LIN {X 0,Y 229.274,Z 915.624,A -85,B 0,C 180,E1 -19873.985,E2 -19873.985} C_VEL
LIN {X 0,Y 228.055,Z 917.353,A -85,B 0,C 180,E1 -19875.727,E2 -19875.727} C_VEL
LIN {X 0,Y 226.593,Z 919.668,A -85,B 0,C 180,E1 -19879.275,E2 -19879.275} C_VEL
LIN {X 0,Y 225.973,Z 920.566,A -85,B 0,C 180,E1 -19882.854,E2 -19882.854} C_VEL
LIN {X 0,Y 225.976,Z 920.476,A -85,B 0,C 180,E1 -19884.646,E2 -19884.646} C_VEL
LIN {X 0,Y 225.996,Z 919.977,A -85,B 0,C 180,E1 -19886.434,E2 -19886.434} C_VEL
LIN {X 0,Y 226.528,Z 918.616,A -85,B 0,C 180,E1 -19889.222,E2 -19889.222} C_VEL
LIN {X 0,Y 226.128,Z 920.542,A -85,B 0,C 180,E1 -19891.781,E2 -19891.781} C_VEL
LIN {X 0,Y 225.942,Z 921.419,A -85,B 0,C 180,E1 -19893.567,E2 -19893.567} C_VEL
LIN {X 0,Y 225.888,Z 921.89,A -85,B 0,C 180,E1 -19895.356,E2 -19895.356} C_VEL
LIN {X 0,Y 226.143,Z 921.695,A -85,B 0,C 180,E1 -19898.939,E2 -19898.939} C_VEL
LIN {X 0,Y 227.195,Z 920.074,A -85,B 0,C 180,E1 -19902.506,E2 -19902.506} C_VEL
LIN {X 0,Y 229.242,Z 917.045,A -85,B 0,C 180,E1 -19906.017,E2 -19906.017} C_VEL
LIN {X 0,Y 232.33,Z 912.52,A -85,B 0,C 180,E1 -19909.436,E2 -19909.436} C_VEL
LIN {X 0,Y 235.463,Z 907.702,A -85,B 0,C 180,E1 -19912.195,E2 -19912.195} C_VEL
LIN {X 0,Y 240.567,Z 900.015,A -85,B 0,C 180,E1 -19915.526,E2 -19915.526} C_VEL
LIN {X 0,Y 245.79,Z 891.995,A -85,B 0,C 180,E1 -19918.151,E2 -19918.151} C_VEL
LIN {X 0,Y 250.12,Z 884.192,A -85,B 0,C 180,E1 -19920.383,E2 -19920.383} C_VEL
LIN {X 0,Y 252.409,Z 878.686,A -85,B 0,C 180,E1 -19921.94,E2 -19921.94} C_VEL
LIN {X 0,Y 254.404,Z 871.949,A -85,B 0,C 180,E1 -19924.026,E2 -19924.026} C_VEL
LIN {X 0,Y 255.766,Z 865.461,A -85,B 0,C 180,E1 -19926.236,E2 -19926.236} C_VEL
LIN {X 0,Y 256.678,Z 859.986,A -85,B 0,C 180,E1 -19928.36,E2 -19928.36} C_VEL
LIN {X 0,Y 257.141,Z 856.349,A -85,B 0,C 180,E1 -19930.066,E2 -19930.066} C_VEL
LIN {X 0,Y 257.235,Z 854.79,A -85,B 0,C 180,E1 -19930.974,E2 -19930.974} C_VEL
LIN {X 0,Y 257.299,Z 852.156,A -85,B 0,C 180,E1 -19933.068,E2 -19933.068} C_VEL
LIN {X 0,Y 257.511,Z 850.333,A -85,B 0,C 180,E1 -19935.202,E2 -19935.202} C_VEL
LIN {X 0,Y 257.586,Z 849.784,A -85,B 0,C 180,E1 -19937.449,E2 -19937.449} C_VEL
LIN {X 0,Y 257.795,Z 850.294,A -85,B 0,C 180,E1 -19939.759,E2 -19939.759} C_VEL
LIN {X 0,Y 258.353,Z 851.607,A -85,B 0,C 180,E1 -19942.082,E2 -19942.082} C_VEL
LIN {X 0,Y 258.93,Z 854.139,A -85,B 0,C 180,E1 -19944.516,E2 -19944.516} C_VEL
LIN {X 0,Y 259.161,Z 858.452,A -85,B 0,C 180,E1 -19947.211,E2 -19947.211} C_VEL
LIN {X 0,Y 258.966,Z 861.924,A -85,B 0,C 180,E1 -19948.958,E2 -19948.958} C_VEL
LIN {X 0,Y 258.495,Z 863.102,A -85,B 0,C 180,E1 -19949.349,E2 -19949.349} C_VEL
LIN {X 0,Y 253.364,Z 871.191,A -85,B 0,C 180,E1 -19951.411,E2 -19951.411} C_VEL
LIN {X 0,Y 247.771,Z 879.009,A -85,B 0,C 180,E1 -19953.916,E2 -19953.916} C_VEL
LIN {X 0,Y 243.503,Z 884.513,A -85,B 0,C 180,E1 -19956.166,E2 -19956.166} C_VEL
LIN {X 0,Y 238.668,Z 890.302,A -85,B 0,C 180,E1 -19959.305,E2 -19959.305} C_VEL
LIN {X 0,Y 234.541,Z 894.493,A -85,B 0,C 180,E1 -19962.562,E2 -19962.562} C_VEL
LIN {X 0,Y 231.301,Z 897.237,A -85,B 0,C 180,E1 -19965.93,E2 -19965.93} C_VEL
LIN {X 0,Y 228.992,Z 898.506,A -85,B 0,C 180,E1 -19969.387,E2 -19969.387} C_VEL
LIN {X 0,Y 227.917,Z 898.617,A -85,B 0,C 180,E1 -19971.129,E2 -19971.129} C_VEL
LIN {X 0,Y 226.816,Z 897.718,A -85,B 0,C 180,E1 -19974.665,E2 -19974.665} C_VEL
LIN {X 0,Y 226.441,Z 896.735,A -85,B 0,C 180,E1 -19976.439,E2 -19976.439} C_VEL
LIN {X 0,Y 226.012,Z 893.548,A -85,B 0,C 180,E1 -19979.998,E2 -19979.998} C_VEL
LIN {X 0,Y 225.989,Z 890.103,A -85,B 0,C 180,E1 -19982.672,E2 -19982.672} C_VEL
LIN {X 0,Y 226.162,Z 884.293,A -85,B 0,C 180,E1 -19986.062,E2 -19986.062} C_VEL
LIN {X 0,Y 226.666,Z 877.901,A -85,B 0,C 180,E1 -19988.917,E2 -19988.917} C_VEL
LIN {X 0,Y 227.604,Z 869.128,A -85,B 0,C 180,E1 -19992.028,E2 -19992.028} C_VEL
LIN {X 0,Y 228.751,Z 859.802,A -85,B 0,C 180,E1 -19994.681,E2 -19994.681} C_VEL
LIN {X 0,Y 230.145,Z 849.412,A -85,B 0,C 180,E1 -19997.091,E2 -19997.091} C_VEL
LIN {X 0,Y 231.52,Z 839.174,A -85,B 0,C 180,E1 -19999.044,E2 -19999.044} C_VEL
LIN {X 0,Y 232.891,Z 827.155,A -85,B 0,C 180,E1 -20000.897,E2 -20000.897} C_VEL
LIN {X 0,Y 230.637,Z 814.342,A -85,B 0,C 180,E1 -20002.616,E2 -20002.616} C_VEL
LIN {X 0,Y 228.031,Z 800.57,A -85,B 0,C 180,E1 -20004.085,E2 -20004.085} C_VEL
LIN {X 0,Y 226.663,Z 793.254,A -85,B 0,C 180,E1 -20004.743,E2 -20004.743} C_VEL
LIN {X 0,Y 227.192,Z 793.184,A -85,B 0,C 180,E1 -20009.984,E2 -20009.984} C_VEL
LIN {X 0,Y 227.538,Z 793.139,A -85,B 0,C 180,E1 -20013.775,E2 -20013.775} C_VEL
LIN {X 0,Y 227.764,Z 793.114,A -85,B 0,C 180,E1 -20016.652,E2 -20016.652} C_VEL
LIN {X 0,Y 227.804,Z 793.107,A -85,B 0,C 180,E1 -20020.379,E2 -20020.379} C_VEL
LIN {X 0,Y 227.82,Z 793.106,A -85,B 0,C 180,E1 -20025.193,E2 -20025.193} C_VEL
LIN {X 0,Y 227.819,Z 793.102,A -85,B 0,C 180,E1 -20029.622,E2 -20029.622} C_VEL
LIN {X 0,Y 227.874,Z 793.098,A -85,B 0,C 180,E1 -20034.127,E2 -20034.127} C_VEL
LIN {X 0,Y 227.849,Z 793.098,A -85,B 0,C 180,E1 -20038.374,E2 -20038.374} C_VEL
LIN {X 0,Y 227.848,Z 793.101,A -85,B 0,C 180,E1 -20042.44,E2 -20042.44} C_VEL
LIN {X 0,Y 227.887,Z 793.094,A -85,B 0,C 180,E1 -20046.364,E2 -20046.364} C_VEL
LIN {X 0,Y 227.906,Z 793.094,A -85,B 0,C 180,E1 -20050.171,E2 -20050.171} C_VEL
LIN {X 0,Y 228.012,Z 793.081,A -85,B 0,C 180,E1 -20053.894,E2 -20053.894} C_VEL
LIN {X 0,Y 228.056,Z 793.075,A -85,B 0,C 180,E1 -20057.542,E2 -20057.542} C_VEL
LIN {X 0,Y 228.249,Z 793.052,A -85,B 0,C 180,E1 -20061.144,E2 -20061.144} C_VEL
LIN {X 0,Y 228.296,Z 793.045,A -85,B 0,C 180,E1 -20062.927,E2 -20062.927} C_VEL
LIN {X 0,Y 228.524,Z 793.019,A -85,B 0,C 180,E1 -20068.238,E2 -20068.238} C_VEL
LIN {X 0,Y 228.522,Z 793.019,A -85,B 0,C 180,E1 -20071.762,E2 -20071.762} C_VEL
LIN {X 0,Y 228.295,Z 793.045,A -85,B 0,C 180,E1 -20077.073,E2 -20077.073} C_VEL
LIN {X 0,Y 228.131,Z 793.066,A -85,B 0,C 180,E1 -20080.652,E2 -20080.652} C_VEL
LIN {X 0,Y 228.025,Z 793.079,A -85,B 0,C 180,E1 -20084.275,E2 -20084.275} C_VEL
LIN {X 0,Y 227.943,Z 793.09,A -85,B 0,C 180,E1 -20087.958,E2 -20087.958} C_VEL
LIN {X 0,Y 227.912,Z 793.093,A -85,B 0,C 180,E1 -20092.323,E2 -20092.323} C_VEL
LIN {X 0,Y 227.915,Z 793.096,A -85,B 0,C 180,E1 -20096.593,E2 -20096.593} C_VEL
LIN {X 0,Y 227.866,Z 793.098,A -85,B 0,C 180,E1 -20100.282,E2 -20100.282} C_VEL
LIN {X 0,Y 227.87,Z 793.098,A -85,B 0,C 180,E1 -20103.722,E2 -20103.722} C_VEL
LIN {X 0,Y 227.838,Z 793.101,A -85,B 0,C 180,E1 -20108.093,E2 -20108.093} C_VEL
LIN {X 0,Y 227.8,Z 793.107,A -85,B 0,C 180,E1 -20112.745,E2 -20112.745} C_VEL
LIN {X 0,Y 227.801,Z 793.11,A -85,B 0,C 180,E1 -20117.258,E2 -20117.258} C_VEL
LIN {X 0,Y 227.819,Z 793.105,A -85,B 0,C 180,E1 -20121.907,E2 -20121.907} C_VEL
LIN {X 0,Y 227.769,Z 793.111,A -85,B 0,C 180,E1 -20124.11,E2 -20124.11} C_VEL
LIN {X 0,Y 227.434,Z 793.149,A -85,B 0,C 180,E1 -20128.313,E2 -20128.313} C_VEL
LIN {X 0,Y 226.937,Z 793.215,A -85,B 0,C 180,E1 -20132.322,E2 -20132.322} C_VEL
LIN {X 0,Y 226.654,Z 793.252,A -85,B 0,C 180,E1 -20135.553,E2 -20135.553} C_VEL
LIN {X 0,Y 229.321,Z 806.969,A -85,B 0,C 180,E1 -20136.84,E2 -20136.84} C_VEL
LIN {X 0,Y 231.8,Z 820.663,A -85,B 0,C 180,E1 -20138.474,E2 -20138.474} C_VEL
LIN {X 0,Y 232.666,Z 825.324,A -85,B 0,C 180,E1 -20139.122,E2 -20139.122} C_VEL
LIN {X 0,Y 231.979,Z 833.383,A -85,B 0,C 180,E1 -20140.297,E2 -20140.297} C_VEL
LIN {X 0,Y 230.728,Z 843.502,A -85,B 0,C 180,E1 -20142.039,E2 -20142.039} C_VEL
LIN {X 0,Y 229.496,Z 853.032,A -85,B 0,C 180,E1 -20144.003,E2 -20144.003} C_VEL
LIN {X 0,Y 228.137,Z 863.503,A -85,B 0,C 180,E1 -20146.643,E2 -20146.643} C_VEL
LIN {X 0,Y 227.143,Z 872.111,A -85,B 0,C 180,E1 -20149.303,E2 -20149.303} C_VEL
LIN {X 0,Y 226.404,Z 880.147,A -85,B 0,C 180,E1 -20152.421,E2 -20152.421} C_VEL
LIN {X 0,Y 225.98,Z 886.444,A -85,B 0,C 180,E1 -20155.543,E2 -20155.543} C_VEL
LIN {X 0,Y 225.964,Z 890.617,A -85,B 0,C 180,E1 -20158.22,E2 -20158.22} C_VEL
LIN {X 0,Y 226.118,Z 894.632,A -85,B 0,C 180,E1 -20161.783,E2 -20161.783} C_VEL
LIN {X 0,Y 226.385,Z 896.062,A -85,B 0,C 180,E1 -20163.562,E2 -20163.562} C_VEL
LIN {X 0,Y 227.142,Z 897.716,A -85,B 0,C 180,E1 -20167.111,E2 -20167.111} C_VEL
LIN {X 0,Y 227.829,Z 897.994,A -85,B 0,C 180,E1 -20168.874,E2 -20168.874} C_VEL
LIN {X 0,Y 229.973,Z 897.451,A -85,B 0,C 180,E1 -20172.354,E2 -20172.354} C_VEL
LIN {X 0,Y 231.14,Z 896.64,A -85,B 0,C 180,E1 -20174.08,E2 -20174.08} C_VEL
LIN {X 0,Y 234.297,Z 893.909,A -85,B 0,C 180,E1 -20177.457,E2 -20177.457} C_VEL
LIN {X 0,Y 237.348,Z 890.881,A -85,B 0,C 180,E1 -20179.91,E2 -20179.91} C_VEL
LIN {X 0,Y 242.013,Z 885.458,A -85,B 0,C 180,E1 -20183.083,E2 -20183.083} C_VEL
LIN {X 0,Y 246.059,Z 880.284,A -85,B 0,C 180,E1 -20185.37,E2 -20185.37} C_VEL
LIN {X 0,Y 252.248,Z 871.669,A -85,B 0,C 180,E1 -20188.273,E2 -20188.273} C_VEL
LIN {X 0,Y 257.284,Z 863.741,A -85,B 0,C 180,E1 -20190.356,E2 -20190.356} C_VEL
LIN {X 0,Y 259.094,Z 860.814,A -85,B 0,C 180,E1 -20191.024,E2 -20191.024} C_VEL
LIN {X 0,Y 259.55,Z 858.602,A -85,B 0,C 180,E1 -20191.9,E2 -20191.9} C_VEL
LIN {X 0,Y 259.84,Z 853.152,A -85,B 0,C 180,E1 -20194.612,E2 -20194.612} C_VEL
LIN {X 0,Y 259.696,Z 850.208,A -85,B 0,C 180,E1 -20196.541,E2 -20196.541} C_VEL
LIN {X 0,Y 259.34,Z 848.043,A -85,B 0,C 180,E1 -20198.558,E2 -20198.558} C_VEL
LIN {X 0,Y 258.983,Z 846.706,A -85,B 0,C 180,E1 -20200.64,E2 -20200.64} C_VEL
LIN {X 0,Y 258.907,Z 846.038,A -85,B 0,C 180,E1 -20202.869,E2 -20202.869} C_VEL
LIN {X 0,Y 258.908,Z 846.524,A -85,B 0,C 180,E1 -20205.108,E2 -20205.108} C_VEL
LIN {X 0,Y 258.887,Z 848.218,A -85,B 0,C 180,E1 -20207.26,E2 -20207.26} C_VEL
LIN {X 0,Y 259.001,Z 850.946,A -85,B 0,C 180,E1 -20209.447,E2 -20209.447} C_VEL
LIN {X 0,Y 258.848,Z 853.067,A -85,B 0,C 180,E1 -20210.528,E2 -20210.528} C_VEL
LIN {X 0,Y 257.691,Z 857.975,A -85,B 0,C 180,E1 -20212.273,E2 -20212.273} C_VEL
LIN {X 0,Y 257.305,Z 859.517,A -85,B 0,C 180,E1 -20212.775,E2 -20212.775} C_VEL
LIN {X 0,Y 256.461,Z 861.959,A -85,B 0,C 180,E1 -20213.454,E2 -20213.454} C_VEL
LIN {X 0,Y 253.775,Z 867.478,A -85,B 0,C 180,E1 -20214.607,E2 -20214.607} C_VEL
LIN {X 0,Y 248.764,Z 875.735,A -85,B 0,C 180,E1 -20216.227,E2 -20216.227} C_VEL
LIN {X 0,Y 246.672,Z 879.511,A -85,B 0,C 180,E1 -20217.167,E2 -20217.167} C_VEL
LIN {X 0,Y 246.146,Z 880.683,A -85,B 0,C 180,E1 -20217.516,E2 -20217.516} C_VEL
LIN {X 0,Y 241.237,Z 889.819,A -85,B 0,C 180,E1 -20220.313,E2 -20220.313} C_VEL
LIN {X 0,Y 235.114,Z 898.779,A -85,B 0,C 180,E1 -20223.36,E2 -20223.36} C_VEL
LIN {X 0,Y 229.931,Z 905.805,A -85,B 0,C 180,E1 -20226.491,E2 -20226.491} C_VEL
LIN {X 0,Y 226.613,Z 910.344,A -85,B 0,C 180,E1 -20229.105,E2 -20229.105} C_VEL
LIN {X 0,Y 223.982,Z 913.873,A -85,B 0,C 180,E1 -20231.713,E2 -20231.713} C_VEL
LIN {X 0,Y 221.163,Z 917.308,A -85,B 0,C 180,E1 -20235.273,E2 -20235.273} C_VEL
LIN {X 0,Y 219.602,Z 919.371,A -85,B 0,C 180,E1 -20238.929,E2 -20238.929} C_VEL
LIN {X 0,Y 218.913,Z 919.999,A -85,B 0,C 180,E1 -20242.622,E2 -20242.622} C_VEL
LIN {X 0,Y 218.931,Z 919.755,A -85,B 0,C 180,E1 -20244.474,E2 -20244.474} C_VEL
LIN {X 0,Y 219.283,Z 918.157,A -85,B 0,C 180,E1 -20248.163,E2 -20248.163} C_VEL
LIN {X 0,Y 219.509,Z 917.46,A -85,B 0,C 180,E1 -20249.197,E2 -20249.197} C_VEL
LIN {X 0,Y 219.501,Z 918.235,A -85,B 0,C 180,E1 -20250,E2 -20250} C_VEL
LIN {X 0,Y 218.887,Z 920.572,A -85,B 0,C 180,E1 -20253.682,E2 -20253.682} C_VEL
LIN {X 0,Y 218.826,Z 921.166,A -85,B 0,C 180,E1 -20255.529,E2 -20255.529} C_VEL
LIN {X 0,Y 219.117,Z 921.256,A -85,B 0,C 180,E1 -20259.228,E2 -20259.228} C_VEL
LIN {X 0,Y 220.224,Z 919.881,A -85,B 0,C 180,E1 -20262.908,E2 -20262.908} C_VEL
LIN {X 0,Y 222.421,Z 917.134,A -85,B 0,C 180,E1 -20266.522,E2 -20266.522} C_VEL
LIN {X 0,Y 225.655,Z 913.026,A -85,B 0,C 180,E1 -20270.035,E2 -20270.035} C_VEL
LIN {X 0,Y 228.919,Z 908.548,A -85,B 0,C 180,E1 -20272.828,E2 -20272.828} C_VEL
LIN {X 0,Y 233.583,Z 902.247,A -85,B 0,C 180,E1 -20275.866,E2 -20275.866} C_VEL
LIN {X 0,Y 239.709,Z 893.799,A -85,B 0,C 180,E1 -20278.932,E2 -20278.932} C_VEL
LIN {X 0,Y 244.314,Z 886.391,A -85,B 0,C 180,E1 -20281.184,E2 -20281.184} C_VEL
LIN {X 0,Y 246.853,Z 881.322,A -85,B 0,C 180,E1 -20282.748,E2 -20282.748} C_VEL
LIN {X 0,Y 249.39,Z 874.036,A -85,B 0,C 180,E1 -20285.188,E2 -20285.188} C_VEL
LIN {X 0,Y 251.014,Z 867.959,A -85,B 0,C 180,E1 -20287.482,E2 -20287.482} C_VEL
LIN {X 0,Y 252.24,Z 862.597,A -85,B 0,C 180,E1 -20289.854,E2 -20289.854} C_VEL
LIN {X 0,Y 252.646,Z 860.025,A -85,B 0,C 180,E1 -20291.314,E2 -20291.314} C_VEL
LIN {X 0,Y 252.907,Z 857.226,A -85,B 0,C 180,E1 -20293.736,E2 -20293.736} C_VEL
LIN {X 0,Y 253.184,Z 855.661,A -85,B 0,C 180,E1 -20296.197,E2 -20296.197} C_VEL
LIN {X 0,Y 253.275,Z 855.58,A -85,B 0,C 180,E1 -20298.522,E2 -20298.522} C_VEL
LIN {X 0,Y 253.6,Z 856.404,A -85,B 0,C 180,E1 -20300.893,E2 -20300.893} C_VEL
LIN {X 0,Y 253.997,Z 858.254,A -85,B 0,C 180,E1 -20303.362,E2 -20303.362} C_VEL
LIN {X 0,Y 254.112,Z 860.071,A -85,B 0,C 180,E1 -20304.942,E2 -20304.942} C_VEL
LIN {X 0,Y 253.822,Z 864.506,A -85,B 0,C 180,E1 -20307.704,E2 -20307.704} C_VEL
LIN {X 0,Y 253.671,Z 865.547,A -85,B 0,C 180,E1 -20308.236,E2 -20308.236} C_VEL
LIN {X 0,Y 251.11,Z 869.408,A -85,B 0,C 180,E1 -20309.283,E2 -20309.283} C_VEL
LIN {X 0,Y 244.171,Z 878.647,A -85,B 0,C 180,E1 -20312.112,E2 -20312.112} C_VEL
LIN {X 0,Y 238.725,Z 885.068,A -85,B 0,C 180,E1 -20314.729,E2 -20314.729} C_VEL
LIN {X 0,Y 234.702,Z 889.543,A -85,B 0,C 180,E1 -20317.089,E2 -20317.089} C_VEL
LIN {X 0,Y 229.966,Z 894.111,A -85,B 0,C 180,E1 -20320.354,E2 -20320.354} C_VEL
LIN {X 0,Y 226.128,Z 897.232,A -85,B 0,C 180,E1 -20323.755,E2 -20323.755} C_VEL
LIN {X 0,Y 223.19,Z 898.882,A -85,B 0,C 180,E1 -20327.264,E2 -20327.264} C_VEL
LIN {X 0,Y 220.939,Z 899.166,A -85,B 0,C 180,E1 -20330.847,E2 -20330.847} C_VEL
LIN {X 0,Y 219.752,Z 897.979,A -85,B 0,C 180,E1 -20334.492,E2 -20334.492} C_VEL
LIN {X 0,Y 219.082,Z 895.308,A -85,B 0,C 180,E1 -20338.16,E2 -20338.16} C_VEL
LIN {X 0,Y 218.914,Z 892.292,A -85,B 0,C 180,E1 -20340.918,E2 -20340.918} C_VEL
LIN {X 0,Y 218.944,Z 888.294,A -85,B 0,C 180,E1 -20343.679,E2 -20343.679} C_VEL
LIN {X 0,Y 219.174,Z 882.707,A -85,B 0,C 180,E1 -20346.697,E2 -20346.697} C_VEL
LIN {X 0,Y 219.742,Z 875.83,A -85,B 0,C 180,E1 -20349.664,E2 -20349.664} C_VEL
LIN {X 0,Y 220.652,Z 867.913,A -85,B 0,C 180,E1 -20352.413,E2 -20352.413} C_VEL
LIN {X 0,Y 221.853,Z 858.216,A -85,B 0,C 180,E1 -20355.148,E2 -20355.148} C_VEL
LIN {X 0,Y 223.167,Z 848.457,A -85,B 0,C 180,E1 -20357.406,E2 -20357.406} C_VEL
LIN {X 0,Y 224.565,Z 837.878,A -85,B 0,C 180,E1 -20359.42,E2 -20359.42} C_VEL
LIN {X 0,Y 225.74,Z 828.36,A -85,B 0,C 180,E1 -20360.933,E2 -20360.933} C_VEL
LIN {X 0,Y 225.16,Z 823.7,A -85,B 0,C 180,E1 -20361.618,E2 -20361.618} C_VEL
LIN {X 0,Y 222.678,Z 810.2,A -85,B 0,C 180,E1 -20363.362,E2 -20363.362} C_VEL
LIN {X 0,Y 219.831,Z 795.12,A -85,B 0,C 180,E1 -20364.882,E2 -20364.882} C_VEL
LIN {X 0,Y 219.649,Z 794.127,A -85,B 0,C 180,E1 -20364.987,E2 -20364.987} C_VEL
LIN {X 0,Y 220.183,Z 794.055,A -85,B 0,C 180,E1 -20370.479,E2 -20370.479} C_VEL
LIN {X 0,Y 220.579,Z 794.008,A -85,B 0,C 180,E1 -20374.993,E2 -20374.993} C_VEL
LIN {X 0,Y 220.733,Z 793.987,A -85,B 0,C 180,E1 -20377.251,E2 -20377.251} C_VEL
LIN {X 0,Y 220.768,Z 793.982,A -85,B 0,C 180,E1 -20380.179,E2 -20380.179} C_VEL
LIN {X 0,Y 220.762,Z 793.986,A -85,B 0,C 180,E1 -20384.454,E2 -20384.454} C_VEL
LIN {X 0,Y 220.761,Z 793.982,A -85,B 0,C 180,E1 -20388.045,E2 -20388.045} C_VEL
LIN {X 0,Y 220.8,Z 793.977,A -85,B 0,C 180,E1 -20390.462,E2 -20390.462} C_VEL
LIN {X 0,Y 220.794,Z 793.983,A -85,B 0,C 180,E1 -20395.044,E2 -20395.044} C_VEL
LIN {X 0,Y 220.827,Z 793.976,A -85,B 0,C 180,E1 -20399.388,E2 -20399.388} C_VEL
LIN {X 0,Y 220.868,Z 793.972,A -85,B 0,C 180,E1 -20403.546,E2 -20403.546} C_VEL
LIN {X 0,Y 220.859,Z 793.971,A -85,B 0,C 180,E1 -20407.551,E2 -20407.551} C_VEL
LIN {X 0,Y 220.921,Z 793.964,A -85,B 0,C 180,E1 -20412.617,E2 -20412.617} C_VEL
LIN {X 0,Y 220.993,Z 793.952,A -85,B 0,C 180,E1 -20417.137,E2 -20417.137} C_VEL
LIN {X 0,Y 221.188,Z 793.931,A -85,B 0,C 180,E1 -20420.859,E2 -20420.859} C_VEL
LIN {X 0,Y 221.234,Z 793.924,A -85,B 0,C 180,E1 -20422.7,E2 -20422.7} C_VEL
LIN {X 0,Y 221.458,Z 793.899,A -85,B 0,C 180,E1 -20428.181,E2 -20428.181} C_VEL
LIN {X 0,Y 221.455,Z 793.9,A -85,B 0,C 180,E1 -20431.819,E2 -20431.819} C_VEL
LIN {X 0,Y 221.232,Z 793.924,A -85,B 0,C 180,E1 -20437.3,E2 -20437.3} C_VEL
LIN {X 0,Y 221.052,Z 793.947,A -85,B 0,C 180,E1 -20440.997,E2 -20440.997} C_VEL
LIN {X 0,Y 220.97,Z 793.961,A -85,B 0,C 180,E1 -20446.633,E2 -20446.633} C_VEL
LIN {X 0,Y 220.863,Z 793.974,A -85,B 0,C 180,E1 -20450.489,E2 -20450.489} C_VEL
LIN {X 0,Y 220.84,Z 793.974,A -85,B 0,C 180,E1 -20454.438,E2 -20454.438} C_VEL
LIN {X 0,Y 220.797,Z 793.982,A -85,B 0,C 180,E1 -20458.519,E2 -20458.519} C_VEL
LIN {X 0,Y 220.805,Z 793.978,A -85,B 0,C 180,E1 -20462.758,E2 -20462.758} C_VEL
LIN {X 0,Y 220.804,Z 793.98,A -85,B 0,C 180,E1 -20467.279,E2 -20467.279} C_VEL
LIN {X 0,Y 220.789,Z 793.977,A -85,B 0,C 180,E1 -20470.19,E2 -20470.19} C_VEL
LIN {X 0,Y 220.762,Z 793.984,A -85,B 0,C 180,E1 -20474.457,E2 -20474.457} C_VEL
LIN {X 0,Y 220.761,Z 793.982,A -85,B 0,C 180,E1 -20478.048,E2 -20478.048} C_VEL
LIN {X 0,Y 220.782,Z 793.981,A -85,B 0,C 180,E1 -20482.787,E2 -20482.787} C_VEL
LIN {X 0,Y 220.45,Z 794.023,A -85,B 0,C 180,E1 -20487.185,E2 -20487.185} C_VEL
LIN {X 0,Y 220.261,Z 794.045,A -85,B 0,C 180,E1 -20489.486,E2 -20489.486} C_VEL
LIN {X 0,Y 219.602,Z 794.128,A -85,B 0,C 180,E1 -20495.165,E2 -20495.165} C_VEL
LIN {X 0,Y 219.616,Z 794.127,A -85,B 0,C 180,E1 -20495.324,E2 -20495.324} C_VEL
LIN {X 0,Y 222.387,Z 808.353,A -85,B 0,C 180,E1 -20496.733,E2 -20496.733} C_VEL
LIN {X 0,Y 224.688,Z 821.078,A -85,B 0,C 180,E1 -20498.311,E2 -20498.311} C_VEL
LIN {X 0,Y 225.648,Z 826.797,A -85,B 0,C 180,E1 -20499.128,E2 -20499.128} C_VEL
LIN {X 0,Y 224.175,Z 839.996,A -85,B 0,C 180,E1 -20501.258,E2 -20501.258} C_VEL
LIN {X 0,Y 222.664,Z 851.133,A -85,B 0,C 180,E1 -20503.499,E2 -20503.499} C_VEL
LIN {X 0,Y 221.206,Z 862.094,A -85,B 0,C 180,E1 -20506.217,E2 -20506.217} C_VEL
LIN {X 0,Y 220.165,Z 870.982,A -85,B 0,C 180,E1 -20508.96,E2 -20508.96} C_VEL
LIN {X 0,Y 219.47,Z 878.246,A -85,B 0,C 180,E1 -20511.717,E2 -20511.717} C_VEL
LIN {X 0,Y 218.994,Z 884.18,A -85,B 0,C 180,E1 -20514.477,E2 -20514.477} C_VEL
LIN {X 0,Y 218.884,Z 888.955,A -85,B 0,C 180,E1 -20517.241,E2 -20517.241} C_VEL
LIN {X 0,Y 218.907,Z 892.674,A -85,B 0,C 180,E1 -20520.002,E2 -20520.002} C_VEL
LIN {X 0,Y 219.304,Z 896.122,A -85,B 0,C 180,E1 -20523.677,E2 -20523.677} C_VEL
LIN {X 0,Y 220.121,Z 898.108,A -85,B 0,C 180,E1 -20527.339,E2 -20527.339} C_VEL
LIN {X 0,Y 220.861,Z 898.528,A -85,B 0,C 180,E1 -20529.157,E2 -20529.157} C_VEL
LIN {X 0,Y 223.082,Z 898.252,A -85,B 0,C 180,E1 -20532.742,E2 -20532.742} C_VEL
LIN {X 0,Y 225.932,Z 896.617,A -85,B 0,C 180,E1 -20536.26,E2 -20536.26} C_VEL
LIN {X 0,Y 227.673,Z 895.256,A -85,B 0,C 180,E1 -20537.982,E2 -20537.982} C_VEL
LIN {X 0,Y 232.029,Z 891.365,A -85,B 0,C 180,E1 -20541.315,E2 -20541.315} C_VEL
LIN {X 0,Y 235.758,Z 887.484,A -85,B 0,C 180,E1 -20543.732,E2 -20543.732} C_VEL
LIN {X 0,Y 239.99,Z 882.66,A -85,B 0,C 180,E1 -20546.059,E2 -20546.059} C_VEL
LIN {X 0,Y 245.599,Z 875.726,A -85,B 0,C 180,E1 -20548.642,E2 -20548.642} C_VEL
LIN {X 0,Y 251.649,Z 867.293,A -85,B 0,C 180,E1 -20551.11,E2 -20551.11} C_VEL
LIN {X 0,Y 253.516,Z 864.526,A -85,B 0,C 180,E1 -20551.786,E2 -20551.786} C_VEL
LIN {X 0,Y 254.186,Z 863.241,A -85,B 0,C 180,E1 -20552.173,E2 -20552.173} C_VEL
LIN {X 0,Y 254.792,Z 859.432,A -85,B 0,C 180,E1 -20554.157,E2 -20554.157} C_VEL
LIN {X 0,Y 255.049,Z 855.815,A -85,B 0,C 180,E1 -20556.518,E2 -20556.518} C_VEL
LIN {X 0,Y 254.812,Z 853.129,A -85,B 0,C 180,E1 -20559.441,E2 -20559.441} C_VEL
LIN {X 0,Y 254.667,Z 852.04,A -85,B 0,C 180,E1 -20561.831,E2 -20561.831} C_VEL
LIN {X 0,Y 254.676,Z 851.984,A -85,B 0,C 180,E1 -20564.152,E2 -20564.152} C_VEL
LIN {X 0,Y 254.607,Z 853.265,A -85,B 0,C 180,E1 -20566.363,E2 -20566.363} C_VEL
LIN {X 0,Y 254.625,Z 855.468,A -85,B 0,C 180,E1 -20568.514,E2 -20568.514} C_VEL
LIN {X 0,Y 254.291,Z 857.874,A -85,B 0,C 180,E1 -20569.943,E2 -20569.943} C_VEL
LIN {X 0,Y 252.312,Z 864.065,A -85,B 0,C 180,E1 -20572.208,E2 -20572.208} C_VEL
LIN {X 0,Y 250.105,Z 870.62,A -85,B 0,C 180,E1 -20574.381,E2 -20574.381} C_VEL
LIN {X 0,Y 246.554,Z 879.693,A -85,B 0,C 180,E1 -20577.208,E2 -20577.208} C_VEL
LIN {X 0,Y 246.146,Z 880.683,A -85,B 0,C 180,E1 -20577.516,E2 -20577.516} C_VEL
LIN {X 0,Y 244.869,Z 883.063,A -85,B 0,C 180,E1 -20578.183,E2 -20578.183} C_VEL
LIN {X 0,Y 243.058,Z 885.529,A -85,B 0,C 180,E1 -20578.769,E2 -20578.769} C_VEL
LIN {X 0,Y 238.497,Z 890.44,A -85,B 0,C 180,E1 -20579.802,E2 -20579.802} C_VEL
LIN {X 0,Y 232.457,Z 896.222,A -85,B 0,C 180,E1 -20581.171,E2 -20581.171} C_VEL
LIN {X 0,Y 229.592,Z 899.271,A -85,B 0,C 180,E1 -20582.227,E2 -20582.227} C_VEL
LIN {X 0,Y 224.68,Z 905.316,A -85,B 0,C 180,E1 -20585.022,E2 -20585.022} C_VEL
LIN {X 0,Y 220.004,Z 910.911,A -85,B 0,C 180,E1 -20588.447,E2 -20588.447} C_VEL
LIN {X 0,Y 217.249,Z 914.141,A -85,B 0,C 180,E1 -20591.125,E2 -20591.125} C_VEL
LIN {X 0,Y 214.291,Z 917.274,A -85,B 0,C 180,E1 -20594.789,E2 -20594.789} C_VEL
LIN {X 0,Y 212.609,Z 919,A -85,B 0,C 180,E1 -20598.56,E2 -20598.56} C_VEL
LIN {X 0,Y 211.879,Z 919.346,A -85,B 0,C 180,E1 -20602.376,E2 -20602.376} C_VEL
LIN {X 0,Y 211.897,Z 919.004,A -85,B 0,C 180,E1 -20604.29,E2 -20604.29} C_VEL
LIN {X 0,Y 211.894,Z 918.269,A -85,B 0,C 180,E1 -20606.196,E2 -20606.196} C_VEL
LIN {X 0,Y 212.498,Z 916.413,A -85,B 0,C 180,E1 -20609.289,E2 -20609.289} C_VEL
LIN {X 0,Y 212.063,Z 918.6,A -85,B 0,C 180,E1 -20611.899,E2 -20611.899} C_VEL
LIN {X 0,Y 211.769,Z 920.388,A -85,B 0,C 180,E1 -20615.714,E2 -20615.714} C_VEL
LIN {X 0,Y 212.108,Z 920.715,A -85,B 0,C 180,E1 -20619.536,E2 -20619.536} C_VEL
LIN {X 0,Y 213.268,Z 919.651,A -85,B 0,C 180,E1 -20623.337,E2 -20623.337} C_VEL
LIN {X 0,Y 215.621,Z 917.237,A -85,B 0,C 180,E1 -20627.059,E2 -20627.059} C_VEL
LIN {X 0,Y 218.999,Z 913.416,A -85,B 0,C 180,E1 -20630.671,E2 -20630.671} C_VEL
LIN {X 0,Y 222.105,Z 909.711,A -85,B 0,C 180,E1 -20633.299,E2 -20633.299} C_VEL
LIN {X 0,Y 227.304,Z 903.404,A -85,B 0,C 180,E1 -20636.636,E2 -20636.636} C_VEL
LIN {X 0,Y 232.804,Z 896.597,A -85,B 0,C 180,E1 -20639.378,E2 -20639.378} C_VEL
LIN {X 0,Y 237.777,Z 889.813,A -85,B 0,C 180,E1 -20641.644,E2 -20641.644} C_VEL
LIN {X 0,Y 240.69,Z 884.993,A -85,B 0,C 180,E1 -20643.195,E2 -20643.195} C_VEL
LIN {X 0,Y 243.59,Z 878.502,A -85,B 0,C 180,E1 -20645.512,E2 -20645.512} C_VEL
LIN {X 0,Y 245.561,Z 872.98,A -85,B 0,C 180,E1 -20647.7,E2 -20647.7} C_VEL
LIN {X 0,Y 247.071,Z 868.272,A -85,B 0,C 180,E1 -20649.821,E2 -20649.821} C_VEL
LIN {X 0,Y 247.957,Z 864.793,A -85,B 0,C 180,E1 -20651.905,E2 -20651.905} C_VEL
LIN {X 0,Y 248.132,Z 863.688,A -85,B 0,C 180,E1 -20652.826,E2 -20652.826} C_VEL
LIN {X 0,Y 248.44,Z 861.824,A -85,B 0,C 180,E1 -20655.009,E2 -20655.009} C_VEL
LIN {X 0,Y 248.62,Z 861.016,A -85,B 0,C 180,E1 -20657.305,E2 -20657.305} C_VEL
LIN {X 0,Y 248.747,Z 861.33,A -85,B 0,C 180,E1 -20659.716,E2 -20659.716} C_VEL
LIN {X 0,Y 249,Z 862.533,A -85,B 0,C 180,E1 -20662.214,E2 -20662.214} C_VEL
LIN {X 0,Y 249.099,Z 863.804,A -85,B 0,C 180,E1 -20663.665,E2 -20663.665} C_VEL
LIN {X 0,Y 248.865,Z 866.18,A -85,B 0,C 180,E1 -20665.61,E2 -20665.61} C_VEL
LIN {X 0,Y 248.318,Z 869.042,A -85,B 0,C 180,E1 -20667.468,E2 -20667.468} C_VEL
LIN {X 0,Y 241.815,Z 877.299,A -85,B 0,C 180,E1 -20669.909,E2 -20669.909} C_VEL
LIN {X 0,Y 235.784,Z 884.066,A -85,B 0,C 180,E1 -20672.482,E2 -20672.482} C_VEL
LIN {X 0,Y 231.136,Z 888.806,A -85,B 0,C 180,E1 -20674.804,E2 -20674.804} C_VEL
LIN {X 0,Y 225.847,Z 893.726,A -85,B 0,C 180,E1 -20678.071,E2 -20678.071} C_VEL
LIN {X 0,Y 221.296,Z 897.141,A -85,B 0,C 180,E1 -20681.481,E2 -20681.481} C_VEL
LIN {X 0,Y 217.712,Z 899.197,A -85,B 0,C 180,E1 -20685.032,E2 -20685.032} C_VEL
LIN {X 0,Y 215.105,Z 899.85,A -85,B 0,C 180,E1 -20688.693,E2 -20688.693} C_VEL
LIN {X 0,Y 213.172,Z 899.079,A -85,B 0,C 180,E1 -20692.42,E2 -20692.42} C_VEL
LIN {X 0,Y 212.301,Z 896.889,A -85,B 0,C 180,E1 -20696.202,E2 -20696.202} C_VEL
LIN {X 0,Y 211.911,Z 894.237,A -85,B 0,C 180,E1 -20699.048,E2 -20699.048} C_VEL
LIN {X 0,Y 211.825,Z 890.69,A -85,B 0,C 180,E1 -20701.899,E2 -20701.899} C_VEL
LIN {X 0,Y 211.867,Z 885.787,A -85,B 0,C 180,E1 -20704.954,E2 -20704.954} C_VEL
LIN {X 0,Y 212.358,Z 879.394,A -85,B 0,C 180,E1 -20708.084,E2 -20708.084} C_VEL
LIN {X 0,Y 213.202,Z 870.803,A -85,B 0,C 180,E1 -20711.405,E2 -20711.405} C_VEL
LIN {X 0,Y 214.276,Z 861.752,A -85,B 0,C 180,E1 -20714.238,E2 -20714.238} C_VEL
LIN {X 0,Y 215.83,Z 850.651,A -85,B 0,C 180,E1 -20717.039,E2 -20717.039} C_VEL
LIN {X 0,Y 217.38,Z 839.211,A -85,B 0,C 180,E1 -20719.351,E2 -20719.351} C_VEL
LIN {X 0,Y 218.675,Z 827.665,A -85,B 0,C 180,E1 -20721.246,E2 -20721.246} C_VEL
LIN {X 0,Y 216.347,Z 814.921,A -85,B 0,C 180,E1 -20723.058,E2 -20723.058} C_VEL
LIN {X 0,Y 213.742,Z 800.789,A -85,B 0,C 180,E1 -20724.672,E2 -20724.672} C_VEL
LIN {X 0,Y 212.626,Z 795.001,A -85,B 0,C 180,E1 -20725.251,E2 -20725.251} C_VEL
LIN {X 0,Y 213.175,Z 794.925,A -85,B 0,C 180,E1 -20730.999,E2 -20730.999} C_VEL
LIN {X 0,Y 213.513,Z 794.89,A -85,B 0,C 180,E1 -20734.624,E2 -20734.624} C_VEL
LIN {X 0,Y 213.669,Z 794.868,A -85,B 0,C 180,E1 -20738.676,E2 -20738.676} C_VEL
LIN {X 0,Y 213.698,Z 794.862,A -85,B 0,C 180,E1 -20741.126,E2 -20741.126} C_VEL
LIN {X 0,Y 213.698,Z 794.863,A -85,B 0,C 180,E1 -20743.678,E2 -20743.678} C_VEL
LIN {X 0,Y 213.698,Z 794.865,A -85,B 0,C 180,E1 -20746.343,E2 -20746.343} C_VEL
LIN {X 0,Y 213.711,Z 794.861,A -85,B 0,C 180,E1 -20749.142,E2 -20749.142} C_VEL
LIN {X 0,Y 213.737,Z 794.859,A -85,B 0,C 180,E1 -20753.71,E2 -20753.71} C_VEL
LIN {X 0,Y 213.752,Z 794.853,A -85,B 0,C 180,E1 -20758.26,E2 -20758.26} C_VEL
LIN {X 0,Y 213.781,Z 794.854,A -85,B 0,C 180,E1 -20762.597,E2 -20762.597} C_VEL
LIN {X 0,Y 213.803,Z 794.85,A -85,B 0,C 180,E1 -20766.978,E2 -20766.978} C_VEL
LIN {X 0,Y 213.884,Z 794.841,A -85,B 0,C 180,E1 -20772.799,E2 -20772.799} C_VEL
LIN {X 0,Y 213.932,Z 794.83,A -85,B 0,C 180,E1 -20776.705,E2 -20776.705} C_VEL
LIN {X 0,Y 214.127,Z 794.81,A -85,B 0,C 180,E1 -20780.555,E2 -20780.555} C_VEL
LIN {X 0,Y 214.065,Z 794.816,A -85,B 0,C 180,E1 -20784.348,E2 -20784.348} C_VEL
LIN {X 0,Y 214.395,Z 794.78,A -85,B 0,C 180,E1 -20788.121,E2 -20788.121} C_VEL
LIN {X 0,Y 214.502,Z 794.768,A -85,B 0,C 180,E1 -20790,E2 -20790} C_VEL
LIN {X 0,Y 214.392,Z 794.78,A -85,B 0,C 180,E1 -20791.879,E2 -20791.879} C_VEL
LIN {X 0,Y 214.173,Z 794.804,A -85,B 0,C 180,E1 -20797.542,E2 -20797.542} C_VEL
LIN {X 0,Y 213.983,Z 794.827,A -85,B 0,C 180,E1 -20801.365,E2 -20801.365} C_VEL
LIN {X 0,Y 213.891,Z 794.838,A -85,B 0,C 180,E1 -20805.24,E2 -20805.24} C_VEL
LIN {X 0,Y 213.803,Z 794.851,A -85,B 0,C 180,E1 -20809.191,E2 -20809.191} C_VEL
LIN {X 0,Y 213.795,Z 794.85,A -85,B 0,C 180,E1 -20813.233,E2 -20813.233} C_VEL
LIN {X 0,Y 213.779,Z 794.854,A -85,B 0,C 180,E1 -20817.429,E2 -20817.429} C_VEL
LIN {X 0,Y 213.752,Z 794.853,A -85,B 0,C 180,E1 -20821.74,E2 -20821.74} C_VEL
LIN {X 0,Y 213.737,Z 794.859,A -85,B 0,C 180,E1 -20826.29,E2 -20826.29} C_VEL
LIN {X 0,Y 213.705,Z 794.862,A -85,B 0,C 180,E1 -20831.127,E2 -20831.127} C_VEL
LIN {X 0,Y 213.698,Z 794.865,A -85,B 0,C 180,E1 -20833.681,E2 -20833.681} C_VEL
LIN {X 0,Y 213.698,Z 794.863,A -85,B 0,C 180,E1 -20836.347,E2 -20836.347} C_VEL
LIN {X 0,Y 213.707,Z 794.863,A -85,B 0,C 180,E1 -20839.147,E2 -20839.147} C_VEL
LIN {X 0,Y 213.657,Z 794.871,A -85,B 0,C 180,E1 -20843.697,E2 -20843.697} C_VEL
LIN {X 0,Y 213.516,Z 794.886,A -85,B 0,C 180,E1 -20845.977,E2 -20845.977} C_VEL
LIN {X 0,Y 213.062,Z 794.942,A -85,B 0,C 180,E1 -20850.347,E2 -20850.347} C_VEL
LIN {X 0,Y 212.572,Z 795.004,A -85,B 0,C 180,E1 -20855.076,E2 -20855.076} C_VEL
LIN {X 0,Y 215.162,Z 808.246,A -85,B 0,C 180,E1 -20856.443,E2 -20856.443} C_VEL
LIN {X 0,Y 217.593,Z 821.633,A -85,B 0,C 180,E1 -20858.161,E2 -20858.161} C_VEL
LIN {X 0,Y 218.532,Z 827.825,A -85,B 0,C 180,E1 -20859.083,E2 -20859.083} C_VEL
LIN {X 0,Y 216.907,Z 841.253,A -85,B 0,C 180,E1 -20861.342,E2 -20861.342} C_VEL
LIN {X 0,Y 215.549,Z 851.208,A -85,B 0,C 180,E1 -20863.426,E2 -20863.426} C_VEL
LIN {X 0,Y 214.088,Z 862.138,A -85,B 0,C 180,E1 -20866.234,E2 -20866.234} C_VEL
LIN {X 0,Y 213.043,Z 871.042,A -85,B 0,C 180,E1 -20869.068,E2 -20869.068} C_VEL
LIN {X 0,Y 212.354,Z 878.383,A -85,B 0,C 180,E1 -20871.916,E2 -20871.916} C_VEL
LIN {X 0,Y 211.821,Z 885.176,A -85,B 0,C 180,E1 -20875.193,E2 -20875.193} C_VEL
LIN {X 0,Y 211.787,Z 889.879,A -85,B 0,C 180,E1 -20878.1,E2 -20878.1} C_VEL
LIN {X 0,Y 211.982,Z 894.468,A -85,B 0,C 180,E1 -20881.902,E2 -20881.902} C_VEL
LIN {X 0,Y 212.226,Z 896.176,A -85,B 0,C 180,E1 -20883.799,E2 -20883.799} C_VEL
LIN {X 0,Y 213.087,Z 898.392,A -85,B 0,C 180,E1 -20887.583,E2 -20887.583} C_VEL
LIN {X 0,Y 215.018,Z 899.186,A -85,B 0,C 180,E1 -20891.312,E2 -20891.312} C_VEL
LIN {X 0,Y 217.54,Z 898.557,A -85,B 0,C 180,E1 -20894.98,E2 -20894.98} C_VEL
LIN {X 0,Y 221.054,Z 896.509,A -85,B 0,C 180,E1 -20898.54,E2 -20898.54} C_VEL
LIN {X 0,Y 225.632,Z 893.064,A -85,B 0,C 180,E1 -20901.951,E2 -20901.951} C_VEL
LIN {X 0,Y 230.933,Z 888.108,A -85,B 0,C 180,E1 -20905.22,E2 -20905.22} C_VEL
LIN {X 0,Y 235.539,Z 883.307,A -85,B 0,C 180,E1 -20907.55,E2 -20907.55} C_VEL
LIN {X 0,Y 241.547,Z 876.51,A -85,B 0,C 180,E1 -20910.128,E2 -20910.128} C_VEL
LIN {X 0,Y 248.029,Z 868.186,A -85,B 0,C 180,E1 -20912.575,E2 -20912.575} C_VEL
LIN {X 0,Y 248.943,Z 866.915,A -85,B 0,C 180,E1 -20912.921,E2 -20912.921} C_VEL
LIN {X 0,Y 249.902,Z 862.807,A -85,B 0,C 180,E1 -20915.356,E2 -20915.356} C_VEL
LIN {X 0,Y 250.231,Z 860.689,A -85,B 0,C 180,E1 -20916.94,E2 -20916.94} C_VEL
LIN {X 0,Y 250.18,Z 859.544,A -85,B 0,C 180,E1 -20918.173,E2 -20918.173} C_VEL
LIN {X 0,Y 250.176,Z 858.019,A -85,B 0,C 180,E1 -20920.669,E2 -20920.669} C_VEL
LIN {X 0,Y 250.259,Z 857.489,A -85,B 0,C 180,E1 -20923.1,E2 -20923.1} C_VEL
LIN {X 0,Y 250.214,Z 858.218,A -85,B 0,C 180,E1 -20925.396,E2 -20925.396} C_VEL
LIN {X 0,Y 250.095,Z 860.03,A -85,B 0,C 180,E1 -20927.59,E2 -20927.59} C_VEL
LIN {X 0,Y 249.95,Z 861.303,A -85,B 0,C 180,E1 -20928.597,E2 -20928.597} C_VEL
LIN {X 0,Y 249.406,Z 863.146,A -85,B 0,C 180,E1 -20929.6,E2 -20929.6} C_VEL
LIN {X 0,Y 246.104,Z 871.281,A -85,B 0,C 180,E1 -20932.639,E2 -20932.639} C_VEL
LIN {X 0,Y 242.2,Z 879.959,A -85,B 0,C 180,E1 -20935.577,E2 -20935.577} C_VEL
LIN {X 0,Y 239.011,Z 885.904,A -85,B 0,C 180,E1 -20937.545,E2 -20937.545} C_VEL
LIN {X 0,Y 233.693,Z 893.97,A -85,B 0,C 180,E1 -20940.25,E2 -20940.25} C_VEL
LIN {X 0,Y 229.592,Z 899.271,A -85,B 0,C 180,E1 -20942.227,E2 -20942.227} C_VEL
LIN {X 0,Y 226.808,Z 902.135,A -85,B 0,C 180,E1 -20943.336,E2 -20943.336} C_VEL
LIN {X 0,Y 220.87,Z 906.522,A -85,B 0,C 180,E1 -20945.045,E2 -20945.045} C_VEL
LIN {X 0,Y 215.172,Z 910.217,A -85,B 0,C 180,E1 -20946.919,E2 -20946.919} C_VEL
LIN {X 0,Y 212.816,Z 912.036,A -85,B 0,C 180,E1 -20948.265,E2 -20948.265} C_VEL
LIN {X 0,Y 208.865,Z 915.918,A -85,B 0,C 180,E1 -20952.372,E2 -20952.372} C_VEL
LIN {X 0,Y 206.362,Z 918.027,A -85,B 0,C 180,E1 -20956.208,E2 -20956.208} C_VEL
LIN {X 0,Y 205.095,Z 918.806,A -85,B 0,C 180,E1 -20960.134,E2 -20960.134} C_VEL
LIN {X 0,Y 204.861,Z 918.116,A -85,B 0,C 180,E1 -20964.216,E2 -20964.216} C_VEL
LIN {X 0,Y 205.247,Z 916.071,A -85,B 0,C 180,E1 -20968.038,E2 -20968.038} C_VEL
LIN {X 0,Y 205.525,Z 915.157,A -85,B 0,C 180,E1 -20969.265,E2 -20969.265} C_VEL
LIN {X 0,Y 205.068,Z 917.487,A -85,B 0,C 180,E1 -20971.964,E2 -20971.964} C_VEL
LIN {X 0,Y 204.73,Z 919.557,A -85,B 0,C 180,E1 -20975.911,E2 -20975.911} C_VEL
LIN {X 0,Y 205.088,Z 920.157,A -85,B 0,C 180,E1 -20979.866,E2 -20979.866} C_VEL
LIN {X 0,Y 206.33,Z 919.355,A -85,B 0,C 180,E1 -20983.794,E2 -20983.794} C_VEL
LIN {X 0,Y 208.844,Z 917.24,A -85,B 0,C 180,E1 -20987.63,E2 -20987.63} C_VEL
LIN {X 0,Y 212.376,Z 913.823,A -85,B 0,C 180,E1 -20991.347,E2 -20991.347} C_VEL
LIN {X 0,Y 216.965,Z 909.055,A -85,B 0,C 180,E1 -20994.904,E2 -20994.904} C_VEL
LIN {X 0,Y 222.608,Z 902.851,A -85,B 0,C 180,E1 -20998.266,E2 -20998.266} C_VEL
LIN {X 0,Y 229.457,Z 895.131,A -85,B 0,C 180,E1 -21001.379,E2 -21001.379} C_VEL
LIN {X 0,Y 234.402,Z 888.482,A -85,B 0,C 180,E1 -21003.689,E2 -21003.689} C_VEL
LIN {X 0,Y 236.925,Z 884.069,A -85,B 0,C 180,E1 -21005.341,E2 -21005.341} C_VEL
LIN {X 0,Y 239.627,Z 878.428,A -85,B 0,C 180,E1 -21007.636,E2 -21007.636} C_VEL
LIN {X 0,Y 242.029,Z 872.538,A -85,B 0,C 180,E1 -21010.425,E2 -21010.425} C_VEL
LIN {X 0,Y 243.118,Z 869.229,A -85,B 0,C 180,E1 -21012.645,E2 -21012.645} C_VEL
LIN {X 0,Y 243.346,Z 868.038,A -85,B 0,C 180,E1 -21013.879,E2 -21013.879} C_VEL
LIN {X 0,Y 243.656,Z 866.635,A -85,B 0,C 180,E1 -21016.189,E2 -21016.189} C_VEL
LIN {X 0,Y 243.789,Z 866.344,A -85,B 0,C 180,E1 -21018.55,E2 -21018.55} C_VEL
LIN {X 0,Y 243.913,Z 867.015,A -85,B 0,C 180,E1 -21021.075,E2 -21021.075} C_VEL
LIN {X 0,Y 243.948,Z 868.045,A -85,B 0,C 180,E1 -21022.77,E2 -21022.77} C_VEL
LIN {X 0,Y 243.673,Z 870.014,A -85,B 0,C 180,E1 -21024.77,E2 -21024.77} C_VEL
LIN {X 0,Y 242.928,Z 872.603,A -85,B 0,C 180,E1 -21026.653,E2 -21026.653} C_VEL
LIN {X 0,Y 235.129,Z 881.256,A -85,B 0,C 180,E1 -21029.459,E2 -21029.459} C_VEL
LIN {X 0,Y 229.845,Z 886.539,A -85,B 0,C 180,E1 -21031.708,E2 -21031.708} C_VEL
LIN {X 0,Y 223.54,Z 892.157,A -85,B 0,C 180,E1 -21034.883,E2 -21034.883} C_VEL
LIN {X 0,Y 219.444,Z 895.342,A -85,B 0,C 180,E1 -21037.397,E2 -21037.397} C_VEL
LIN {X 0,Y 214.703,Z 898.44,A -85,B 0,C 180,E1 -21040.891,E2 -21040.891} C_VEL
LIN {X 0,Y 210.935,Z 900.097,A -85,B 0,C 180,E1 -21044.539,E2 -21044.539} C_VEL
LIN {X 0,Y 208.17,Z 900.411,A -85,B 0,C 180,E1 -21048.311,E2 -21048.311} C_VEL
LIN {X 0,Y 206.142,Z 899.367,A -85,B 0,C 180,E1 -21052.16,E2 -21052.16} C_VEL
LIN {X 0,Y 205.225,Z 896.847,A -85,B 0,C 180,E1 -21056.071,E2 -21056.071} C_VEL
LIN {X 0,Y 204.798,Z 892.854,A -85,B 0,C 180,E1 -21059.998,E2 -21059.998} C_VEL
LIN {X 0,Y 204.749,Z 888.736,A -85,B 0,C 180,E1 -21062.949,E2 -21062.949} C_VEL
LIN {X 0,Y 204.9,Z 883.572,A -85,B 0,C 180,E1 -21065.904,E2 -21065.904} C_VEL
LIN {X 0,Y 205.398,Z 877.247,A -85,B 0,C 180,E1 -21068.855,E2 -21068.855} C_VEL
LIN {X 0,Y 206.244,Z 869.476,A -85,B 0,C 180,E1 -21071.796,E2 -21071.796} C_VEL
LIN {X 0,Y 207.388,Z 859.977,A -85,B 0,C 180,E1 -21074.722,E2 -21074.722} C_VEL
LIN {X 0,Y 208.87,Z 849.469,A -85,B 0,C 180,E1 -21077.373,E2 -21077.373} C_VEL
LIN {X 0,Y 210.442,Z 837.758,A -85,B 0,C 180,E1 -21079.761,E2 -21079.761} C_VEL
LIN {X 0,Y 211.505,Z 827.813,A -85,B 0,C 180,E1 -21081.437,E2 -21081.437} C_VEL
LIN {X 0,Y 209.261,Z 815.495,A -85,B 0,C 180,E1 -21083.24,E2 -21083.24} C_VEL
LIN {X 0,Y 206.611,Z 800.915,A -85,B 0,C 180,E1 -21084.952,E2 -21084.952} C_VEL
LIN {X 0,Y 205.579,Z 795.879,A -85,B 0,C 180,E1 -21085.464,E2 -21085.464} C_VEL
LIN {X 0,Y 206.101,Z 795.807,A -85,B 0,C 180,E1 -21090.761,E2 -21090.761} C_VEL
LIN {X 0,Y 206.502,Z 795.76,A -85,B 0,C 180,E1 -21095.347,E2 -21095.347} C_VEL
LIN {X 0,Y 206.635,Z 795.745,A -85,B 0,C 180,E1 -21098.531,E2 -21098.531} C_VEL
LIN {X 0,Y 206.615,Z 795.749,A -85,B 0,C 180,E1 -21102.864,E2 -21102.864} C_VEL
LIN {X 0,Y 206.617,Z 795.746,A -85,B 0,C 180,E1 -21107.133,E2 -21107.133} C_VEL
LIN {X 0,Y 206.682,Z 795.738,A -85,B 0,C 180,E1 -21111.449,E2 -21111.449} C_VEL
LIN {X 0,Y 206.693,Z 795.738,A -85,B 0,C 180,E1 -21114.687,E2 -21114.687} C_VEL
LIN {X 0,Y 206.689,Z 795.737,A -85,B 0,C 180,E1 -21119.333,E2 -21119.333} C_VEL
LIN {X 0,Y 206.698,Z 795.736,A -85,B 0,C 180,E1 -21123.767,E2 -21123.767} C_VEL
LIN {X 0,Y 206.723,Z 795.73,A -85,B 0,C 180,E1 -21128.039,E2 -21128.039} C_VEL
LIN {X 0,Y 206.817,Z 795.721,A -85,B 0,C 180,E1 -21132.191,E2 -21132.191} C_VEL
LIN {X 0,Y 206.871,Z 795.71,A -85,B 0,C 180,E1 -21136.243,E2 -21136.243} C_VEL
LIN {X 0,Y 207.071,Z 795.69,A -85,B 0,C 180,E1 -21140.23,E2 -21140.23} C_VEL
LIN {X 0,Y 207.029,Z 795.693,A -85,B 0,C 180,E1 -21144.155,E2 -21144.155} C_VEL
LIN {X 0,Y 207.334,Z 795.659,A -85,B 0,C 180,E1 -21148.057,E2 -21148.057} C_VEL
LIN {X 0,Y 207.47,Z 795.643,A -85,B 0,C 180,E1 -21150,E2 -21150} C_VEL
LIN {X 0,Y 207.331,Z 795.66,A -85,B 0,C 180,E1 -21151.943,E2 -21151.943} C_VEL
LIN {X 0,Y 207.118,Z 795.684,A -85,B 0,C 180,E1 -21157.801,E2 -21157.801} C_VEL
LIN {X 0,Y 206.906,Z 795.709,A -85,B 0,C 180,E1 -21161.759,E2 -21161.759} C_VEL
LIN {X 0,Y 206.819,Z 795.72,A -85,B 0,C 180,E1 -21165.775,E2 -21165.775} C_VEL
LIN {X 0,Y 206.738,Z 795.731,A -85,B 0,C 180,E1 -21169.874,E2 -21169.874} C_VEL
LIN {X 0,Y 206.731,Z 795.73,A -85,B 0,C 180,E1 -21174.076,E2 -21174.076} C_VEL
LIN {X 0,Y 206.681,Z 795.739,A -85,B 0,C 180,E1 -21178.428,E2 -21178.428} C_VEL
LIN {X 0,Y 206.688,Z 795.737,A -85,B 0,C 180,E1 -21182.96,E2 -21182.96} C_VEL
LIN {X 0,Y 206.673,Z 795.738,A -85,B 0,C 180,E1 -21187.741,E2 -21187.741} C_VEL
LIN {X 0,Y 206.635,Z 795.743,A -85,B 0,C 180,E1 -21191.564,E2 -21191.564} C_VEL
LIN {X 0,Y 206.626,Z 795.746,A -85,B 0,C 180,E1 -21195.584,E2 -21195.584} C_VEL
LIN {X 0,Y 206.648,Z 795.741,A -85,B 0,C 180,E1 -21199.749,E2 -21199.749} C_VEL
LIN {X 0,Y 206.65,Z 795.741,A -85,B 0,C 180,E1 -21202.257,E2 -21202.257} C_VEL
LIN {X 0,Y 206.525,Z 795.757,A -85,B 0,C 180,E1 -21204.757,E2 -21204.757} C_VEL
LIN {X 0,Y 206.168,Z 795.799,A -85,B 0,C 180,E1 -21209.25,E2 -21209.25} C_VEL
LIN {X 0,Y 205.559,Z 795.877,A -85,B 0,C 180,E1 -21214.85,E2 -21214.85} C_VEL
LIN {X 0,Y 208.382,Z 810.451,A -85,B 0,C 180,E1 -21216.451,E2 -21216.451} C_VEL
LIN {X 0,Y 210.75,Z 823.543,A -85,B 0,C 180,E1 -21218.226,E2 -21218.226} C_VEL
LIN {X 0,Y 211.476,Z 827.762,A -85,B 0,C 180,E1 -21218.878,E2 -21218.878} C_VEL
LIN {X 0,Y 209.83,Z 841.049,A -85,B 0,C 180,E1 -21221.195,E2 -21221.195} C_VEL
LIN {X 0,Y 208.452,Z 851.06,A -85,B 0,C 180,E1 -21223.349,E2 -21223.349} C_VEL
LIN {X 0,Y 206.965,Z 862.079,A -85,B 0,C 180,E1 -21226.251,E2 -21226.251} C_VEL
LIN {X 0,Y 205.929,Z 871.104,A -85,B 0,C 180,E1 -21229.183,E2 -21229.183} C_VEL
LIN {X 0,Y 205.209,Z 878.474,A -85,B 0,C 180,E1 -21232.128,E2 -21232.128} C_VEL
LIN {X 0,Y 204.726,Z 884.998,A -85,B 0,C 180,E1 -21235.353,E2 -21235.353} C_VEL
LIN {X 0,Y 204.703,Z 889.367,A -85,B 0,C 180,E1 -21238.035,E2 -21238.035} C_VEL
LIN {X 0,Y 204.812,Z 893.21,A -85,B 0,C 180,E1 -21240.985,E2 -21240.985} C_VEL
LIN {X 0,Y 205.152,Z 896.088,A -85,B 0,C 180,E1 -21243.931,E2 -21243.931} C_VEL
LIN {X 0,Y 206.06,Z 898.658,A -85,B 0,C 180,E1 -21247.843,E2 -21247.843} C_VEL
LIN {X 0,Y 208.094,Z 899.727,A -85,B 0,C 180,E1 -21251.693,E2 -21251.693} C_VEL
LIN {X 0,Y 210.761,Z 899.43,A -85,B 0,C 180,E1 -21255.474,E2 -21255.474} C_VEL
LIN {X 0,Y 214.446,Z 897.783,A -85,B 0,C 180,E1 -21259.133,E2 -21259.133} C_VEL
LIN {X 0,Y 219.234,Z 894.672,A -85,B 0,C 180,E1 -21262.626,E2 -21262.626} C_VEL
LIN {X 0,Y 224.794,Z 890.185,A -85,B 0,C 180,E1 -21265.959,E2 -21265.959} C_VEL
LIN {X 0,Y 229.605,Z 885.8,A -85,B 0,C 180,E1 -21268.325,E2 -21268.325} C_VEL
LIN {X 0,Y 236.76,Z 878.444,A -85,B 0,C 180,E1 -21271.299,E2 -21271.299} C_VEL
LIN {X 0,Y 243.562,Z 870.56,A -85,B 0,C 180,E1 -21273.735,E2 -21273.735} C_VEL
LIN {X 0,Y 244.443,Z 868.286,A -85,B 0,C 180,E1 -21275.103,E2 -21275.103} C_VEL
LIN {X 0,Y 245.156,Z 865.796,A -85,B 0,C 180,E1 -21277.016,E2 -21277.016} C_VEL
LIN {X 0,Y 245.302,Z 864.045,A -85,B 0,C 180,E1 -21279.325,E2 -21279.325} C_VEL
LIN {X 0,Y 245.486,Z 862.985,A -85,B 0,C 180,E1 -21281.896,E2 -21281.896} C_VEL
LIN {X 0,Y 245.596,Z 863.13,A -85,B 0,C 180,E1 -21284.324,E2 -21284.324} C_VEL
LIN {X 0,Y 245.407,Z 864.54,A -85,B 0,C 180,E1 -21286.582,E2 -21286.582} C_VEL
LIN {X 0,Y 245.068,Z 866.274,A -85,B 0,C 180,E1 -21288.215,E2 -21288.215} C_VEL
LIN {X 0,Y 244.191,Z 868.395,A -85,B 0,C 180,E1 -21289.291,E2 -21289.291} C_VEL
LIN {X 0,Y 240.544,Z 875.655,A -85,B 0,C 180,E1 -21292.152,E2 -21292.152} C_VEL
LIN {X 0,Y 236.197,Z 883.638,A -85,B 0,C 180,E1 -21295.056,E2 -21295.056} C_VEL
LIN {X 0,Y 232.575,Z 889.303,A -85,B 0,C 180,E1 -21297.048,E2 -21297.048} C_VEL
LIN {X 0,Y 227.719,Z 895.729,A -85,B 0,C 180,E1 -21299.387,E2 -21299.387} C_VEL
LIN {X 0,Y 221.208,Z 903.163,A -85,B 0,C 180,E1 -21302.569,E2 -21302.569} C_VEL
LIN {X 0,Y 215.795,Z 908.979,A -85,B 0,C 180,E1 -21305.958,E2 -21305.958} C_VEL
LIN {X 0,Y 212.816,Z 912.036,A -85,B 0,C 180,E1 -21308.265,E2 -21308.265} C_VEL
LIN {X 0,Y 210.566,Z 913.685,A -85,B 0,C 180,E1 -21309.679,E2 -21309.679} C_VEL
LIN {X 0,Y 205.475,Z 915.849,A -85,B 0,C 180,E1 -21311.952,E2 -21311.952} C_VEL
LIN {X 0,Y 200.827,Z 917.269,A -85,B 0,C 180,E1 -21314.381,E2 -21314.381} C_VEL
LIN {X 0,Y 199.312,Z 917.75,A -85,B 0,C 180,E1 -21316.004,E2 -21316.004} C_VEL
LIN {X 0,Y 198.091,Z 918.143,A -85,B 0,C 180,E1 -21319.782,E2 -21319.782} C_VEL
LIN {X 0,Y 197.84,Z 917.194,A -85,B 0,C 180,E1 -21324.094,E2 -21324.094} C_VEL
LIN {X 0,Y 198.23,Z 914.904,A -85,B 0,C 180,E1 -21327.968,E2 -21327.968} C_VEL
LIN {X 0,Y 198.543,Z 913.94,A -85,B 0,C 180,E1 -21329.366,E2 -21329.366} C_VEL
LIN {X 0,Y 198.069,Z 916.364,A -85,B 0,C 180,E1 -21332.033,E2 -21332.033} C_VEL
LIN {X 0,Y 197.693,Z 918.627,A -85,B 0,C 180,E1 -21336.122,E2 -21336.122} C_VEL
LIN {X 0,Y 198.084,Z 919.489,A -85,B 0,C 180,E1 -21340.218,E2 -21340.218} C_VEL
LIN {X 0,Y 199.411,Z 919.005,A -85,B 0,C 180,E1 -21344.283,E2 -21344.283} C_VEL
LIN {X 0,Y 202.091,Z 917.238,A -85,B 0,C 180,E1 -21348.239,E2 -21348.239} C_VEL
LIN {X 0,Y 205.786,Z 914.148,A -85,B 0,C 180,E1 -21352.066,E2 -21352.066} C_VEL
LIN {X 0,Y 210.591,Z 909.785,A -85,B 0,C 180,E1 -21355.712,E2 -21355.712} C_VEL
LIN {X 0,Y 216.468,Z 904.08,A -85,B 0,C 180,E1 -21359.144,E2 -21359.144} C_VEL
LIN {X 0,Y 223.583,Z 896.865,A -85,B 0,C 180,E1 -21362.301,E2 -21362.301} C_VEL
LIN {X 0,Y 228.831,Z 890.699,A -85,B 0,C 180,E1 -21364.624,E2 -21364.624} C_VEL
LIN {X 0,Y 231.541,Z 886.6,A -85,B 0,C 180,E1 -21366.291,E2 -21366.291} C_VEL
LIN {X 0,Y 233.82,Z 882.613,A -85,B 0,C 180,E1 -21368.024,E2 -21368.024} C_VEL
LIN {X 0,Y 236.627,Z 877.082,A -85,B 0,C 180,E1 -21370.8,E2 -21370.8} C_VEL
LIN {X 0,Y 237.889,Z 874.159,A -85,B 0,C 180,E1 -21372.804,E2 -21372.804} C_VEL
LIN {X 0,Y 238.383,Z 872.357,A -85,B 0,C 180,E1 -21375.038,E2 -21375.038} C_VEL
LIN {X 0,Y 238.647,Z 871.457,A -85,B 0,C 180,E1 -21377.412,E2 -21377.412} C_VEL
LIN {X 0,Y 238.719,Z 871.588,A -85,B 0,C 180,E1 -21379.948,E2 -21379.948} C_VEL
LIN {X 0,Y 238.685,Z 872.802,A -85,B 0,C 180,E1 -21382.656,E2 -21382.656} C_VEL
LIN {X 0,Y 238.071,Z 874.921,A -85,B 0,C 180,E1 -21384.894,E2 -21384.894} C_VEL
LIN {X 0,Y 237.496,Z 876.061,A -85,B 0,C 180,E1 -21385.787,E2 -21385.787} C_VEL
LIN {X 0,Y 229.439,Z 884.111,A -85,B 0,C 180,E1 -21388.617,E2 -21388.617} C_VEL
LIN {X 0,Y 222.171,Z 890.387,A -85,B 0,C 180,E1 -21391.671,E2 -21391.671} C_VEL
LIN {X 0,Y 215.92,Z 895.121,A -85,B 0,C 180,E1 -21394.965,E2 -21394.965} C_VEL
LIN {X 0,Y 210.489,Z 898.457,A -85,B 0,C 180,E1 -21398.45,E2 -21398.45} C_VEL
LIN {X 0,Y 206.024,Z 900.45,A -85,B 0,C 180,E1 -21402.119,E2 -21402.119} C_VEL
LIN {X 0,Y 202.62,Z 901.115,A -85,B 0,C 180,E1 -21405.946,E2 -21405.946} C_VEL
LIN {X 0,Y 200.006,Z 900.409,A -85,B 0,C 180,E1 -21409.879,E2 -21409.879} C_VEL
LIN {X 0,Y 198.571,Z 898.317,A -85,B 0,C 180,E1 -21413.903,E2 -21413.903} C_VEL
LIN {X 0,Y 197.883,Z 894.797,A -85,B 0,C 180,E1 -21417.963,E2 -21417.963} C_VEL
LIN {X 0,Y 197.704,Z 891.117,A -85,B 0,C 180,E1 -21421.016,E2 -21421.016} C_VEL
LIN {X 0,Y 197.704,Z 885.379,A -85,B 0,C 180,E1 -21424.669,E2 -21424.669} C_VEL
LIN {X 0,Y 198.223,Z 878.008,A -85,B 0,C 180,E1 -21428.316,E2 -21428.316} C_VEL
LIN {X 0,Y 199.134,Z 869.41,A -85,B 0,C 180,E1 -21431.706,E2 -21431.706} C_VEL
LIN {X 0,Y 200.269,Z 859.92,A -85,B 0,C 180,E1 -21434.737,E2 -21434.737} C_VEL
LIN {X 0,Y 201.801,Z 849.284,A -85,B 0,C 180,E1 -21437.478,E2 -21437.478} C_VEL
LIN {X 0,Y 203.397,Z 837.467,A -85,B 0,C 180,E1 -21439.948,E2 -21439.948} C_VEL
LIN {X 0,Y 204.373,Z 828.251,A -85,B 0,C 180,E1 -21441.543,E2 -21441.543} C_VEL
LIN {X 0,Y 202.115,Z 815.872,A -85,B 0,C 180,E1 -21443.422,E2 -21443.422} C_VEL
LIN {X 0,Y 199.577,Z 801.78,A -85,B 0,C 180,E1 -21445.149,E2 -21445.149} C_VEL
LIN {X 0,Y 198.541,Z 796.756,A -85,B 0,C 180,E1 -21445.696,E2 -21445.696} C_VEL
LIN {X 0,Y 198.872,Z 796.71,A -85,B 0,C 180,E1 -21449.651,E2 -21449.651} C_VEL
LIN {X 0,Y 199.159,Z 796.672,A -85,B 0,C 180,E1 -21452.121,E2 -21452.121} C_VEL
LIN {X 0,Y 199.496,Z 796.634,A -85,B 0,C 180,E1 -21456.787,E2 -21456.787} C_VEL
LIN {X 0,Y 199.578,Z 796.62,A -85,B 0,C 180,E1 -21459.332,E2 -21459.332} C_VEL
LIN {X 0,Y 199.564,Z 796.623,A -85,B 0,C 180,E1 -21462.306,E2 -21462.306} C_VEL
LIN {X 0,Y 199.572,Z 796.625,A -85,B 0,C 180,E1 -21465.226,E2 -21465.226} C_VEL
LIN {X 0,Y 199.572,Z 796.622,A -85,B 0,C 180,E1 -21468.003,E2 -21468.003} C_VEL
LIN {X 0,Y 199.604,Z 796.618,A -85,B 0,C 180,E1 -21470.766,E2 -21470.766} C_VEL
LIN {X 0,Y 199.604,Z 796.619,A -85,B 0,C 180,E1 -21475.712,E2 -21475.712} C_VEL
LIN {X 0,Y 199.679,Z 796.606,A -85,B 0,C 180,E1 -21478.133,E2 -21478.133} C_VEL
LIN {X 0,Y 199.636,Z 796.616,A -85,B 0,C 180,E1 -21482.764,E2 -21482.764} C_VEL
LIN {X 0,Y 199.699,Z 796.607,A -85,B 0,C 180,E1 -21487.224,E2 -21487.224} C_VEL
LIN {X 0,Y 199.742,Z 796.604,A -85,B 0,C 180,E1 -21491.798,E2 -21491.798} C_VEL
LIN {X 0,Y 199.808,Z 796.592,A -85,B 0,C 180,E1 -21495.746,E2 -21495.746} C_VEL
LIN {X 0,Y 200.015,Z 796.571,A -85,B 0,C 180,E1 -21499.881,E2 -21499.881} C_VEL
LIN {X 0,Y 199.993,Z 796.57,A -85,B 0,C 180,E1 -21503.948,E2 -21503.948} C_VEL
LIN {X 0,Y 200.276,Z 796.538,A -85,B 0,C 180,E1 -21507.989,E2 -21507.989} C_VEL
LIN {X 0,Y 200.438,Z 796.519,A -85,B 0,C 180,E1 -21510,E2 -21510} C_VEL
LIN {X 0,Y 199.973,Z 796.572,A -85,B 0,C 180,E1 -21514.031,E2 -21514.031} C_VEL
LIN {X 0,Y 200.066,Z 796.564,A -85,B 0,C 180,E1 -21518.078,E2 -21518.078} C_VEL
LIN {X 0,Y 199.856,Z 796.589,A -85,B 0,C 180,E1 -21522.181,E2 -21522.181} C_VEL
LIN {X 0,Y 199.757,Z 796.602,A -85,B 0,C 180,E1 -21526.348,E2 -21526.348} C_VEL
LIN {X 0,Y 199.662,Z 796.613,A -85,B 0,C 180,E1 -21530.61,E2 -21530.61} C_VEL
LIN {X 0,Y 199.643,Z 796.616,A -85,B 0,C 180,E1 -21534.988,E2 -21534.988} C_VEL
LIN {X 0,Y 199.602,Z 796.618,A -85,B 0,C 180,E1 -21539.534,E2 -21539.534} C_VEL
LIN {X 0,Y 199.659,Z 796.609,A -85,B 0,C 180,E1 -21542.354,E2 -21542.354} C_VEL
LIN {X 0,Y 199.617,Z 796.62,A -85,B 0,C 180,E1 -21546.765,E2 -21546.765} C_VEL
LIN {X 0,Y 199.602,Z 796.618,A -85,B 0,C 180,E1 -21549.33,E2 -21549.33} C_VEL
LIN {X 0,Y 199.567,Z 796.622,A -85,B 0,C 180,E1 -21552.311,E2 -21552.311} C_VEL
LIN {X 0,Y 199.572,Z 796.627,A -85,B 0,C 180,E1 -21555.23,E2 -21555.23} C_VEL
LIN {X 0,Y 199.571,Z 796.621,A -85,B 0,C 180,E1 -21558.006,E2 -21558.006} C_VEL
LIN {X 0,Y 199.592,Z 796.618,A -85,B 0,C 180,E1 -21560.774,E2 -21560.774} C_VEL
LIN {X 0,Y 199.49,Z 796.634,A -85,B 0,C 180,E1 -21564.124,E2 -21564.124} C_VEL
LIN {X 0,Y 199.22,Z 796.664,A -85,B 0,C 180,E1 -21568.054,E2 -21568.054} C_VEL
LIN {X 0,Y 198.723,Z 796.729,A -85,B 0,C 180,E1 -21572.631,E2 -21572.631} C_VEL
LIN {X 0,Y 198.538,Z 796.752,A -85,B 0,C 180,E1 -21574.655,E2 -21574.655} C_VEL
LIN {X 0,Y 201.351,Z 811.456,A -85,B 0,C 180,E1 -21576.337,E2 -21576.337} C_VEL
LIN {X 0,Y 203.828,Z 825.117,A -85,B 0,C 180,E1 -21578.291,E2 -21578.291} C_VEL
LIN {X 0,Y 204.34,Z 828.397,A -85,B 0,C 180,E1 -21578.818,E2 -21578.818} C_VEL
LIN {X 0,Y 202.77,Z 840.755,A -85,B 0,C 180,E1 -21581.041,E2 -21581.041} C_VEL
LIN {X 0,Y 201.349,Z 850.895,A -85,B 0,C 180,E1 -21583.266,E2 -21583.266} C_VEL
LIN {X 0,Y 199.847,Z 861.983,A -85,B 0,C 180,E1 -21586.27,E2 -21586.27} C_VEL
LIN {X 0,Y 198.783,Z 871.037,A -85,B 0,C 180,E1 -21589.305,E2 -21589.305} C_VEL
LIN {X 0,Y 197.992,Z 879.574,A -85,B 0,C 180,E1 -21592.865,E2 -21592.865} C_VEL
LIN {X 0,Y 197.652,Z 885.496,A -85,B 0,C 180,E1 -21595.924,E2 -21595.924} C_VEL
LIN {X 0,Y 197.678,Z 890.254,A -85,B 0,C 180,E1 -21598.984,E2 -21598.984} C_VEL
LIN {X 0,Y 197.852,Z 893.974,A -85,B 0,C 180,E1 -21602.038,E2 -21602.038} C_VEL
LIN {X 0,Y 198.081,Z 895.973,A -85,B 0,C 180,E1 -21604.071,E2 -21604.071} C_VEL
LIN {X 0,Y 199.04,Z 898.793,A -85,B 0,C 180,E1 -21608.122,E2 -21608.122} C_VEL
LIN {X 0,Y 201.17,Z 900.222,A -85,B 0,C 180,E1 -21612.102,E2 -21612.102} C_VEL
LIN {X 0,Y 203.998,Z 900.265,A -85,B 0,C 180,E1 -21616,E2 -21616} C_VEL
LIN {X 0,Y 207.853,Z 898.936,A -85,B 0,C 180,E1 -21619.765,E2 -21619.765} C_VEL
LIN {X 0,Y 212.867,Z 896.27,A -85,B 0,C 180,E1 -21623.342,E2 -21623.342} C_VEL
LIN {X 0,Y 218.676,Z 892.215,A -85,B 0,C 180,E1 -21626.742,E2 -21626.742} C_VEL
LIN {X 0,Y 225.458,Z 886.663,A -85,B 0,C 180,E1 -21629.919,E2 -21629.919} C_VEL
LIN {X 0,Y 233.076,Z 879.467,A -85,B 0,C 180,E1 -21632.873,E2 -21632.873} C_VEL
LIN {X 0,Y 238.187,Z 874.123,A -85,B 0,C 180,E1 -21634.612,E2 -21634.612} C_VEL
LIN {X 0,Y 238.757,Z 873.259,A -85,B 0,C 180,E1 -21635.031,E2 -21635.031} C_VEL
LIN {X 0,Y 239.317,Z 872.036,A -85,B 0,C 180,E1 -21635.97,E2 -21635.97} C_VEL
LIN {X 0,Y 240.014,Z 869.996,A -85,B 0,C 180,E1 -21637.947,E2 -21637.947} C_VEL
LIN {X 0,Y 240.363,Z 868.568,A -85,B 0,C 180,E1 -21640.516,E2 -21640.516} C_VEL
LIN {X 0,Y 240.687,Z 868.07,A -85,B 0,C 180,E1 -21643.114,E2 -21643.114} C_VEL
LIN {X 0,Y 240.686,Z 868.393,A -85,B 0,C 180,E1 -21644.493,E2 -21644.493} C_VEL
LIN {X 0,Y 240.59,Z 868.919,A -85,B 0,C 180,E1 -21645.486,E2 -21645.486} C_VEL
LIN {X 0,Y 240.097,Z 870.884,A -85,B 0,C 180,E1 -21647.682,E2 -21647.682} C_VEL
LIN {X 0,Y 238.793,Z 873.306,A -85,B 0,C 180,E1 -21648.911,E2 -21648.911} C_VEL
LIN {X 0,Y 234.935,Z 879.694,A -85,B 0,C 180,E1 -21651.582,E2 -21651.582} C_VEL
LIN {X 0,Y 230.073,Z 887.21,A -85,B 0,C 180,E1 -21654.522,E2 -21654.522} C_VEL
LIN {X 0,Y 225.26,Z 893.493,A -85,B 0,C 180,E1 -21656.907,E2 -21656.907} C_VEL
LIN {X 0,Y 218.274,Z 901.024,A -85,B 0,C 180,E1 -21660.061,E2 -21660.061} C_VEL
LIN {X 0,Y 212.03,Z 907.162,A -85,B 0,C 180,E1 -21663.418,E2 -21663.418} C_VEL
LIN {X 0,Y 206.893,Z 911.878,A -85,B 0,C 180,E1 -21667.005,E2 -21667.005} C_VEL
LIN {X 0,Y 203.826,Z 914.56,A -85,B 0,C 180,E1 -21669.83,E2 -21669.83} C_VEL
LIN {X 0,Y 200.613,Z 916.982,A -85,B 0,C 180,E1 -21673.724,E2 -21673.724} C_VEL
LIN {X 0,Y 199.312,Z 917.75,A -85,B 0,C 180,E1 -21676.004,E2 -21676.004} C_VEL
LIN {X 0,Y 198.023,Z 918.049,A -85,B 0,C 180,E1 -21677.665,E2 -21677.665} C_VEL
LIN {X 0,Y 194.557,Z 917.733,A -85,B 0,C 180,E1 -21680.372,E2 -21680.372} C_VEL
LIN {X 0,Y 191.947,Z 916.856,A -85,B 0,C 180,E1 -21682.59,E2 -21682.59} C_VEL
LIN {X 0,Y 190.895,Z 915.963,A -85,B 0,C 180,E1 -21684.319,E2 -21684.319} C_VEL
LIN {X 0,Y 190.827,Z 915.606,A -85,B 0,C 180,E1 -21684.905,E2 -21684.905} C_VEL
LIN {X 0,Y 191.581,Z 912.551,A -85,B 0,C 180,E1 -21689.343,E2 -21689.343} C_VEL
LIN {X 0,Y 191.083,Z 915.069,A -85,B 0,C 180,E1 -21692.108,E2 -21692.108} C_VEL
LIN {X 0,Y 190.679,Z 917.645,A -85,B 0,C 180,E1 -21696.348,E2 -21696.348} C_VEL
LIN {X 0,Y 191.096,Z 918.784,A -85,B 0,C 180,E1 -21700.596,E2 -21700.596} C_VEL
LIN {X 0,Y 192.514,Z 918.585,A -85,B 0,C 180,E1 -21704.806,E2 -21704.806} C_VEL
LIN {X 0,Y 195.348,Z 917.121,A -85,B 0,C 180,E1 -21708.893,E2 -21708.893} C_VEL
LIN {X 0,Y 199.234,Z 914.418,A -85,B 0,C 180,E1 -21712.832,E2 -21712.832} C_VEL
LIN {X 0,Y 204.264,Z 910.458,A -85,B 0,C 180,E1 -21716.57,E2 -21716.57} C_VEL
LIN {X 0,Y 210.373,Z 905.233,A -85,B 0,C 180,E1 -21720.074,E2 -21720.074} C_VEL
LIN {X 0,Y 217.763,Z 898.561,A -85,B 0,C 180,E1 -21723.275,E2 -21723.275} C_VEL
LIN {X 0,Y 223.276,Z 892.82,A -85,B 0,C 180,E1 -21725.614,E2 -21725.614} C_VEL
LIN {X 0,Y 226.196,Z 889.008,A -85,B 0,C 180,E1 -21727.292,E2 -21727.292} C_VEL
LIN {X 0,Y 228.942,Z 884.863,A -85,B 0,C 180,E1 -21729.317,E2 -21729.317} C_VEL
LIN {X 0,Y 231.704,Z 880.34,A -85,B 0,C 180,E1 -21731.859,E2 -21731.859} C_VEL
LIN {X 0,Y 232.612,Z 878.326,A -85,B 0,C 180,E1 -21733.519,E2 -21733.519} C_VEL
LIN {X 0,Y 233.174,Z 876.614,A -85,B 0,C 180,E1 -21736.334,E2 -21736.334} C_VEL
LIN {X 0,Y 233.332,Z 876.218,A -85,B 0,C 180,E1 -21738.852,E2 -21738.852} C_VEL
LIN {X 0,Y 233.294,Z 876.863,A -85,B 0,C 180,E1 -21741.559,E2 -21741.559} C_VEL
LIN {X 0,Y 233.074,Z 877.607,A -85,B 0,C 180,E1 -21742.908,E2 -21742.908} C_VEL
LIN {X 0,Y 232.118,Z 879.507,A -85,B 0,C 180,E1 -21744.879,E2 -21744.879} C_VEL
LIN {X 0,Y 223.756,Z 886.86,A -85,B 0,C 180,E1 -21747.725,E2 -21747.725} C_VEL
LIN {X 0,Y 218.045,Z 891.3,A -85,B 0,C 180,E1 -21750.025,E2 -21750.025} C_VEL
LIN {X 0,Y 212.805,Z 894.92,A -85,B 0,C 180,E1 -21752.459,E2 -21752.459} C_VEL
LIN {X 0,Y 206.736,Z 898.493,A -85,B 0,C 180,E1 -21755.922,E2 -21755.922} C_VEL
LIN {X 0,Y 201.548,Z 900.784,A -85,B 0,C 180,E1 -21759.59,E2 -21759.59} C_VEL
LIN {X 0,Y 197.407,Z 901.716,A -85,B 0,C 180,E1 -21763.45,E2 -21763.45} C_VEL
LIN {X 0,Y 194.351,Z 901.351,A -85,B 0,C 180,E1 -21767.467,E2 -21767.467} C_VEL
LIN {X 0,Y 192.104,Z 899.657,A -85,B 0,C 180,E1 -21771.583,E2 -21771.583} C_VEL
LIN {X 0,Y 191.084,Z 896.532,A -85,B 0,C 180,E1 -21775.779,E2 -21775.779} C_VEL
LIN {X 0,Y 190.708,Z 893.233,A -85,B 0,C 180,E1 -21778.942,E2 -21778.942} C_VEL
LIN {X 0,Y 190.616,Z 888.984,A -85,B 0,C 180,E1 -21782.111,E2 -21782.111} C_VEL
LIN {X 0,Y 190.756,Z 882.569,A -85,B 0,C 180,E1 -21785.867,E2 -21785.867} C_VEL
LIN {X 0,Y 191.28,Z 875.955,A -85,B 0,C 180,E1 -21788.981,E2 -21788.981} C_VEL
LIN {X 0,Y 192.182,Z 867.792,A -85,B 0,C 180,E1 -21792.136,E2 -21792.136} C_VEL
LIN {X 0,Y 193.414,Z 857.837,A -85,B 0,C 180,E1 -21795.272,E2 -21795.272} C_VEL
LIN {X 0,Y 194.958,Z 846.791,A -85,B 0,C 180,E1 -21798.112,E2 -21798.112} C_VEL
LIN {X 0,Y 196.35,Z 837.172,A -85,B 0,C 180,E1 -21800.149,E2 -21800.149} C_VEL
LIN {X 0,Y 197.324,Z 829.575,A -85,B 0,C 180,E1 -21801.504,E2 -21801.504} C_VEL
LIN {X 0,Y 195.181,Z 817.307,A -85,B 0,C 180,E1 -21803.47,E2 -21803.47} C_VEL
LIN {X 0,Y 192.646,Z 803.149,A -85,B 0,C 180,E1 -21805.294,E2 -21805.294} C_VEL
LIN {X 0,Y 191.53,Z 797.629,A -85,B 0,C 180,E1 -21805.951,E2 -21805.951} C_VEL
LIN {X 0,Y 191.949,Z 797.569,A -85,B 0,C 180,E1 -21810.834,E2 -21810.834} C_VEL
LIN {X 0,Y 192.194,Z 797.541,A -85,B 0,C 180,E1 -21813.262,E2 -21813.262} C_VEL
LIN {X 0,Y 192.461,Z 797.512,A -85,B 0,C 180,E1 -21816.547,E2 -21816.547} C_VEL
LIN {X 0,Y 192.498,Z 797.503,A -85,B 0,C 180,E1 -21821.081,E2 -21821.081} C_VEL
LIN {X 0,Y 192.484,Z 797.507,A -85,B 0,C 180,E1 -21826.074,E2 -21826.074} C_VEL
LIN {X 0,Y 192.511,Z 797.499,A -85,B 0,C 180,E1 -21830.05,E2 -21830.05} C_VEL
LIN {X 0,Y 192.554,Z 797.498,A -85,B 0,C 180,E1 -21834.269,E2 -21834.269} C_VEL
LIN {X 0,Y 192.598,Z 797.492,A -85,B 0,C 180,E1 -21837.059,E2 -21837.059} C_VEL
LIN {X 0,Y 192.613,Z 797.491,A -85,B 0,C 180,E1 -21841.684,E2 -21841.684} C_VEL
LIN {X 0,Y 192.671,Z 797.48,A -85,B 0,C 180,E1 -21846.344,E2 -21846.344} C_VEL
LIN {X 0,Y 192.69,Z 797.484,A -85,B 0,C 180,E1 -21851.487,E2 -21851.487} C_VEL
LIN {X 0,Y 192.733,Z 797.475,A -85,B 0,C 180,E1 -21855.211,E2 -21855.211} C_VEL
LIN {X 0,Y 192.937,Z 797.451,A -85,B 0,C 180,E1 -21859.566,E2 -21859.566} C_VEL
LIN {X 0,Y 192.957,Z 797.448,A -85,B 0,C 180,E1 -21863.727,E2 -21863.727} C_VEL
LIN {X 0,Y 193.221,Z 797.416,A -85,B 0,C 180,E1 -21867.916,E2 -21867.916} C_VEL
LIN {X 0,Y 193.404,Z 797.395,A -85,B 0,C 180,E1 -21870,E2 -21870} C_VEL
LIN {X 0,Y 192.921,Z 797.45,A -85,B 0,C 180,E1 -21874.178,E2 -21874.178} C_VEL
LIN {X 0,Y 193.017,Z 797.443,A -85,B 0,C 180,E1 -21878.375,E2 -21878.375} C_VEL
LIN {X 0,Y 192.782,Z 797.466,A -85,B 0,C 180,E1 -21882.635,E2 -21882.635} C_VEL
LIN {X 0,Y 192.711,Z 797.479,A -85,B 0,C 180,E1 -21886.963,E2 -21886.963} C_VEL
LIN {X 0,Y 192.598,Z 797.489,A -85,B 0,C 180,E1 -21891.402,E2 -21891.402} C_VEL
LIN {X 0,Y 192.632,Z 797.486,A -85,B 0,C 180,E1 -21894.209,E2 -21894.209} C_VEL
LIN {X 0,Y 192.595,Z 797.494,A -85,B 0,C 180,E1 -21898.867,E2 -21898.867} C_VEL
LIN {X 0,Y 192.588,Z 797.495,A -85,B 0,C 180,E1 -21903.188,E2 -21903.188} C_VEL
LIN {X 0,Y 192.545,Z 797.498,A -85,B 0,C 180,E1 -21908.354,E2 -21908.354} C_VEL
LIN {X 0,Y 192.484,Z 797.508,A -85,B 0,C 180,E1 -21913.097,E2 -21913.097} C_VEL
LIN {X 0,Y 192.484,Z 797.508,A -85,B 0,C 180,E1 -21916.907,E2 -21916.907} C_VEL
LIN {X 0,Y 192.492,Z 797.507,A -85,B 0,C 180,E1 -21921.637,E2 -21921.637} C_VEL
LIN {X 0,Y 192.428,Z 797.514,A -85,B 0,C 180,E1 -21924.245,E2 -21924.245} C_VEL
LIN {X 0,Y 192.012,Z 797.561,A -85,B 0,C 180,E1 -21929.177,E2 -21929.177} C_VEL
LIN {X 0,Y 191.52,Z 797.627,A -85,B 0,C 180,E1 -21934.355,E2 -21934.355} C_VEL
LIN {X 0,Y 191.522,Z 797.713,A -85,B 0,C 180,E1 -21934.475,E2 -21934.475} C_VEL
LIN {X 0,Y 194.104,Z 811.265,A -85,B 0,C 180,E1 -21936.06,E2 -21936.06} C_VEL
LIN {X 0,Y 196.415,Z 824.156,A -85,B 0,C 180,E1 -21937.939,E2 -21937.939} C_VEL
LIN {X 0,Y 197.162,Z 828.296,A -85,B 0,C 180,E1 -21938.629,E2 -21938.629} C_VEL
LIN {X 0,Y 195.713,Z 840.407,A -85,B 0,C 180,E1 -21940.875,E2 -21940.875} C_VEL
LIN {X 0,Y 194.143,Z 851.593,A -85,B 0,C 180,E1 -21943.439,E2 -21943.439} C_VEL
LIN {X 0,Y 192.748,Z 861.708,A -85,B 0,C 180,E1 -21946.293,E2 -21946.293} C_VEL
LIN {X 0,Y 191.683,Z 870.91,A -85,B 0,C 180,E1 -21949.439,E2 -21949.439} C_VEL
LIN {X 0,Y 190.985,Z 878.452,A -85,B 0,C 180,E1 -21952.602,E2 -21952.602} C_VEL
LIN {X 0,Y 190.587,Z 884.581,A -85,B 0,C 180,E1 -21955.773,E2 -21955.773} C_VEL
LIN {X 0,Y 190.612,Z 889.594,A -85,B 0,C 180,E1 -21958.946,E2 -21958.946} C_VEL
LIN {X 0,Y 190.789,Z 893.592,A -85,B 0,C 180,E1 -21962.113,E2 -21962.113} C_VEL
LIN {X 0,Y 191.4,Z 897.472,A -85,B 0,C 180,E1 -21966.326,E2 -21966.326} C_VEL
LIN {X 0,Y 192.984,Z 899.939,A -85,B 0,C 180,E1 -21970.493,E2 -21970.493} C_VEL
LIN {X 0,Y 195.625,Z 900.974,A -85,B 0,C 180,E1 -21974.567,E2 -21974.567} C_VEL
LIN {X 0,Y 199.141,Z 900.699,A -85,B 0,C 180,E1 -21978.521,E2 -21978.521} C_VEL
LIN {X 0,Y 201.28,Z 900.082,A -85,B 0,C 180,E1 -21980.438,E2 -21980.438} C_VEL
LIN {X 0,Y 206.534,Z 897.781,A -85,B 0,C 180,E1 -21984.103,E2 -21984.103} C_VEL
LIN {X 0,Y 212.603,Z 894.158,A -85,B 0,C 180,E1 -21987.57,E2 -21987.57} C_VEL
LIN {X 0,Y 217.795,Z 890.526,A -85,B 0,C 180,E1 -21990.013,E2 -21990.013} C_VEL
LIN {X 0,Y 225.543,Z 884.344,A -85,B 0,C 180,E1 -21993.047,E2 -21993.047} C_VEL
LIN {X 0,Y 231.734,Z 878.67,A -85,B 0,C 180,E1 -21995.188,E2 -21995.188} C_VEL
LIN {X 0,Y 233.55,Z 876.781,A -85,B 0,C 180,E1 -21995.932,E2 -21995.932} C_VEL
LIN {X 0,Y 234.102,Z 875.756,A -85,B 0,C 180,E1 -21996.902,E2 -21996.902} C_VEL
LIN {X 0,Y 234.802,Z 874.176,A -85,B 0,C 180,E1 -21998.946,E2 -21998.946} C_VEL
LIN {X 0,Y 235.328,Z 873.112,A -85,B 0,C 180,E1 -22001.701,E2 -22001.701} C_VEL
LIN {X 0,Y 235.559,Z 873.038,A -85,B 0,C 180,E1 -22003.333,E2 -22003.333} C_VEL
LIN {X 0,Y 235.565,Z 873.252,A -85,B 0,C 180,E1 -22004.272,E2 -22004.272} C_VEL
LIN {X 0,Y 235.105,Z 874.769,A -85,B 0,C 180,E1 -22006.564,E2 -22006.564} C_VEL
LIN {X 0,Y 234.261,Z 876.403,A -85,B 0,C 180,E1 -22007.769,E2 -22007.769} C_VEL
LIN {X 0,Y 230.516,Z 881.687,A -85,B 0,C 180,E1 -22010.189,E2 -22010.189} C_VEL
LIN {X 0,Y 226.187,Z 887.561,A -85,B 0,C 180,E1 -22012.706,E2 -22012.706} C_VEL
LIN {X 0,Y 221.302,Z 893.452,A -85,B 0,C 180,E1 -22015.136,E2 -22015.136} C_VEL
LIN {X 0,Y 215.923,Z 899.013,A -85,B 0,C 180,E1 -22017.517,E2 -22017.517} C_VEL
LIN {X 0,Y 208.872,Z 905.33,A -85,B 0,C 180,E1 -22020.798,E2 -22020.798} C_VEL
LIN {X 0,Y 204.063,Z 909.357,A -85,B 0,C 180,E1 -22023.57,E2 -22023.57} C_VEL
LIN {X 0,Y 199.237,Z 913.145,A -85,B 0,C 180,E1 -22027.169,E2 -22027.169} C_VEL
LIN {X 0,Y 195.364,Z 915.845,A -85,B 0,C 180,E1 -22031.109,E2 -22031.109} C_VEL
LIN {X 0,Y 192.542,Z 917.294,A -85,B 0,C 180,E1 -22035.196,E2 -22035.196} C_VEL
LIN {X 0,Y 191.103,Z 917.454,A -85,B 0,C 180,E1 -22039.404,E2 -22039.404} C_VEL
LIN {X 0,Y 190.826,Z 916.128,A -85,B 0,C 180,E1 -22043.946,E2 -22043.946} C_VEL
LIN {X 0,Y 190.827,Z 915.606,A -85,B 0,C 180,E1 -22044.905,E2 -22044.905} C_VEL
LIN {X 0,Y 190.272,Z 914.844,A -85,B 0,C 180,E1 -22046.084,E2 -22046.084} C_VEL
LIN {X 0,Y 187.786,Z 912.984,A -85,B 0,C 180,E1 -22047.948,E2 -22047.948} C_VEL
LIN {X 0,Y 185.144,Z 912.166,A -85,B 0,C 180,E1 -22049.845,E2 -22049.845} C_VEL
LIN {X 0,Y 184.34,Z 912.733,A -85,B 0,C 180,E1 -22051.042,E2 -22051.042} C_VEL
LIN {X 0,Y 183.831,Z 915.358,A -85,B 0,C 180,E1 -22054.385,E2 -22054.385} C_VEL
LIN {X 0,Y 183.793,Z 917.419,A -85,B 0,C 180,E1 -22058.798,E2 -22058.798} C_VEL
LIN {X 0,Y 184.719,Z 918.164,A -85,B 0,C 180,E1 -22063.196,E2 -22063.196} C_VEL
LIN {X 0,Y 187.014,Z 917.67,A -85,B 0,C 180,E1 -22067.496,E2 -22067.496} C_VEL
LIN {X 0,Y 190.526,Z 915.947,A -85,B 0,C 180,E1 -22071.646,E2 -22071.646} C_VEL
LIN {X 0,Y 195.143,Z 913.015,A -85,B 0,C 180,E1 -22075.606,E2 -22075.606} C_VEL
LIN {X 0,Y 201.022,Z 908.831,A -85,B 0,C 180,E1 -22079.305,E2 -22079.305} C_VEL
LIN {X 0,Y 206.166,Z 904.895,A -85,B 0,C 180,E1 -22081.896,E2 -22081.896} C_VEL
LIN {X 0,Y 214.01,Z 898.432,A -85,B 0,C 180,E1 -22085.078,E2 -22085.078} C_VEL
LIN {X 0,Y 217.784,Z 894.836,A -85,B 0,C 180,E1 -22086.656,E2 -22086.656} C_VEL
LIN {X 0,Y 220.876,Z 891.315,A -85,B 0,C 180,E1 -22088.35,E2 -22088.35} C_VEL
LIN {X 0,Y 223.779,Z 887.506,A -85,B 0,C 180,E1 -22090.409,E2 -22090.409} C_VEL
LIN {X 0,Y 225.732,Z 884.867,A -85,B 0,C 180,E1 -22092.019,E2 -22092.019} C_VEL
LIN {X 0,Y 226.671,Z 883.476,A -85,B 0,C 180,E1 -22093.009,E2 -22093.009} C_VEL
LIN {X 0,Y 227.435,Z 881.717,A -85,B 0,C 180,E1 -22095.294,E2 -22095.294} C_VEL
LIN {X 0,Y 227.761,Z 880.852,A -85,B 0,C 180,E1 -22097.78,E2 -22097.78} C_VEL
LIN {X 0,Y 227.754,Z 880.966,A -85,B 0,C 180,E1 -22100.484,E2 -22100.484} C_VEL
LIN {X 0,Y 227.602,Z 881.391,A -85,B 0,C 180,E1 -22101.859,E2 -22101.859} C_VEL
LIN {X 0,Y 226.746,Z 882.801,A -85,B 0,C 180,E1 -22103.919,E2 -22103.919} C_VEL
LIN {X 0,Y 218.122,Z 889.535,A -85,B 0,C 180,E1 -22106.785,E2 -22106.785} C_VEL
LIN {X 0,Y 210.335,Z 894.775,A -85,B 0,C 180,E1 -22109.919,E2 -22109.919} C_VEL
LIN {X 0,Y 203.521,Z 898.547,A -85,B 0,C 180,E1 -22113.324,E2 -22113.324} C_VEL
LIN {X 0,Y 197.587,Z 901.054,A -85,B 0,C 180,E1 -22116.965,E2 -22116.965} C_VEL
LIN {X 0,Y 192.712,Z 902.292,A -85,B 0,C 180,E1 -22120.837,E2 -22120.837} C_VEL
LIN {X 0,Y 188.926,Z 902.236,A -85,B 0,C 180,E1 -22124.904,E2 -22124.904} C_VEL
LIN {X 0,Y 186.05,Z 900.84,A -85,B 0,C 180,E1 -22129.111,E2 -22129.111} C_VEL
LIN {X 0,Y 184.453,Z 898.113,A -85,B 0,C 180,E1 -22133.434,E2 -22133.434} C_VEL
LIN {X 0,Y 183.759,Z 893.974,A -85,B 0,C 180,E1 -22137.806,E2 -22137.806} C_VEL
LIN {X 0,Y 183.572,Z 889.825,A -85,B 0,C 180,E1 -22141.095,E2 -22141.095} C_VEL
LIN {X 0,Y 183.567,Z 884.591,A -85,B 0,C 180,E1 -22144.389,E2 -22144.389} C_VEL
LIN {X 0,Y 184.079,Z 877.014,A -85,B 0,C 180,E1 -22148.229,E2 -22148.229} C_VEL
LIN {X 0,Y 185.08,Z 867.616,A -85,B 0,C 180,E1 -22152.053,E2 -22152.053} C_VEL
LIN {X 0,Y 186.325,Z 857.505,A -85,B 0,C 180,E1 -22155.307,E2 -22155.307} C_VEL
LIN {X 0,Y 187.771,Z 847.416,A -85,B 0,C 180,E1 -22157.984,E2 -22157.984} C_VEL
LIN {X 0,Y 189.314,Z 836.492,A -85,B 0,C 180,E1 -22160.365,E2 -22160.365} C_VEL
LIN {X 0,Y 190.166,Z 829.359,A -85,B 0,C 180,E1 -22161.687,E2 -22161.687} C_VEL
LIN {X 0,Y 187.891,Z 816.9,A -85,B 0,C 180,E1 -22163.725,E2 -22163.725} C_VEL
LIN {X 0,Y 185.172,Z 802.101,A -85,B 0,C 180,E1 -22165.676,E2 -22165.676} C_VEL
LIN {X 0,Y 184.507,Z 798.503,A -85,B 0,C 180,E1 -22166.122,E2 -22166.122} C_VEL
LIN {X 0,Y 184.76,Z 798.468,A -85,B 0,C 180,E1 -22169.634,E2 -22169.634} C_VEL
LIN {X 0,Y 185.246,Z 798.41,A -85,B 0,C 180,E1 -22174.683,E2 -22174.683} C_VEL
LIN {X 0,Y 185.411,Z 798.387,A -85,B 0,C 180,E1 -22177.332,E2 -22177.332} C_VEL
LIN {X 0,Y 185.453,Z 798.38,A -85,B 0,C 180,E1 -22180.718,E2 -22180.718} C_VEL
LIN {X 0,Y 185.453,Z 798.383,A -85,B 0,C 180,E1 -22186.053,E2 -22186.053} C_VEL
LIN {X 0,Y 185.461,Z 798.377,A -85,B 0,C 180,E1 -22189.893,E2 -22189.893} C_VEL
LIN {X 0,Y 185.5,Z 798.377,A -85,B 0,C 180,E1 -22192.71,E2 -22192.71} C_VEL
LIN {X 0,Y 185.524,Z 798.369,A -85,B 0,C 180,E1 -22197.971,E2 -22197.971} C_VEL
LIN {X 0,Y 185.54,Z 798.37,A -85,B 0,C 180,E1 -22200.594,E2 -22200.594} C_VEL
LIN {X 0,Y 185.573,Z 798.368,A -85,B 0,C 180,E1 -22205.38,E2 -22205.38} C_VEL
LIN {X 0,Y 185.626,Z 798.362,A -85,B 0,C 180,E1 -22211.17,E2 -22211.17} C_VEL
LIN {X 0,Y 185.662,Z 798.355,A -85,B 0,C 180,E1 -22214.634,E2 -22214.634} C_VEL
LIN {X 0,Y 185.88,Z 798.33,A -85,B 0,C 180,E1 -22219.418,E2 -22219.418} C_VEL
LIN {X 0,Y 185.922,Z 798.325,A -85,B 0,C 180,E1 -22223.488,E2 -22223.488} C_VEL
LIN {X 0,Y 186.167,Z 798.294,A -85,B 0,C 180,E1 -22227.836,E2 -22227.836} C_VEL
LIN {X 0,Y 186.37,Z 798.272,A -85,B 0,C 180,E1 -22230,E2 -22230} C_VEL
LIN {X 0,Y 185.869,Z 798.328,A -85,B 0,C 180,E1 -22234.337,E2 -22234.337} C_VEL
LIN {X 0,Y 185.966,Z 798.32,A -85,B 0,C 180,E1 -22238.695,E2 -22238.695} C_VEL
LIN {X 0,Y 185.708,Z 798.346,A -85,B 0,C 180,E1 -22243.124,E2 -22243.124} C_VEL
LIN {X 0,Y 185.648,Z 798.358,A -85,B 0,C 180,E1 -22247.629,E2 -22247.629} C_VEL
LIN {X 0,Y 185.562,Z 798.367,A -85,B 0,C 180,E1 -22252.256,E2 -22252.256} C_VEL
LIN {X 0,Y 185.57,Z 798.368,A -85,B 0,C 180,E1 -22254.647,E2 -22254.647} C_VEL
LIN {X 0,Y 185.537,Z 798.37,A -85,B 0,C 180,E1 -22259.501,E2 -22259.501} C_VEL
LIN {X 0,Y 185.492,Z 798.378,A -85,B 0,C 180,E1 -22264.634,E2 -22264.634} C_VEL
LIN {X 0,Y 185.5,Z 798.377,A -85,B 0,C 180,E1 -22267.315,E2 -22267.315} C_VEL
LIN {X 0,Y 185.465,Z 798.378,A -85,B 0,C 180,E1 -22270.726,E2 -22270.726} C_VEL
LIN {X 0,Y 185.453,Z 798.382,A -85,B 0,C 180,E1 -22276.057,E2 -22276.057} C_VEL
LIN {X 0,Y 185.454,Z 798.38,A -85,B 0,C 180,E1 -22279.895,E2 -22279.895} C_VEL
LIN {X 0,Y 185.441,Z 798.384,A -85,B 0,C 180,E1 -22282.738,E2 -22282.738} C_VEL
LIN {X 0,Y 185.186,Z 798.414,A -85,B 0,C 180,E1 -22286.608,E2 -22286.608} C_VEL
LIN {X 0,Y 184.765,Z 798.467,A -85,B 0,C 180,E1 -22291.029,E2 -22291.029} C_VEL
LIN {X 0,Y 184.482,Z 798.504,A -85,B 0,C 180,E1 -22294.268,E2 -22294.268} C_VEL
LIN {X 0,Y 187.469,Z 814.293,A -85,B 0,C 180,E1 -22296.272,E2 -22296.272} C_VEL
LIN {X 0,Y 189.727,Z 826.904,A -85,B 0,C 180,E1 -22298.261,E2 -22298.261} C_VEL
LIN {X 0,Y 190.045,Z 828.781,A -85,B 0,C 180,E1 -22298.584,E2 -22298.584} C_VEL
LIN {X 0,Y 188.673,Z 839.801,A -85,B 0,C 180,E1 -22300.698,E2 -22300.698} C_VEL
LIN {X 0,Y 187.075,Z 851.14,A -85,B 0,C 180,E1 -22303.357,E2 -22303.357} C_VEL
LIN {X 0,Y 185.655,Z 861.435,A -85,B 0,C 180,E1 -22306.317,E2 -22306.317} C_VEL
LIN {X 0,Y 184.714,Z 869.262,A -85,B 0,C 180,E1 -22309.036,E2 -22309.036} C_VEL
LIN {X 0,Y 183.994,Z 877.1,A -85,B 0,C 180,E1 -22312.319,E2 -22312.319} C_VEL
LIN {X 0,Y 183.557,Z 883.573,A -85,B 0,C 180,E1 -22315.611,E2 -22315.611} C_VEL
LIN {X 0,Y 183.547,Z 888.886,A -85,B 0,C 180,E1 -22318.905,E2 -22318.905} C_VEL
LIN {X 0,Y 183.728,Z 893.084,A -85,B 0,C 180,E1 -22322.194,E2 -22322.194} C_VEL
LIN {X 0,Y 184.349,Z 897.307,A -85,B 0,C 180,E1 -22326.569,E2 -22326.569} C_VEL
LIN {X 0,Y 186.022,Z 900.059,A -85,B 0,C 180,E1 -22330.891,E2 -22330.891} C_VEL
LIN {X 0,Y 188.8,Z 901.48,A -85,B 0,C 180,E1 -22335.106,E2 -22335.106} C_VEL
LIN {X 0,Y 192.496,Z 901.563,A -85,B 0,C 180,E1 -22339.185,E2 -22339.185} C_VEL
LIN {X 0,Y 197.357,Z 900.326,A -85,B 0,C 180,E1 -22343.063,E2 -22343.063} C_VEL
LIN {X 0,Y 203.296,Z 897.803,A -85,B 0,C 180,E1 -22346.708,E2 -22346.708} C_VEL
LIN {X 0,Y 210.092,Z 893.971,A -85,B 0,C 180,E1 -22350.12,E2 -22350.12} C_VEL
LIN {X 0,Y 217.899,Z 888.681,A -85,B 0,C 180,E1 -22353.253,E2 -22353.253} C_VEL
LIN {X 0,Y 226.421,Z 881.951,A -85,B 0,C 180,E1 -22356.141,E2 -22356.141} C_VEL
LIN {X 0,Y 228.204,Z 880.326,A -85,B 0,C 180,E1 -22356.8,E2 -22356.8} C_VEL
LIN {X 0,Y 228.779,Z 879.473,A -85,B 0,C 180,E1 -22357.91,E2 -22357.91} C_VEL
LIN {X 0,Y 229.523,Z 878.271,A -85,B 0,C 180,E1 -22360.048,E2 -22360.048} C_VEL
LIN {X 0,Y 230.133,Z 877.744,A -85,B 0,C 180,E1 -22362.867,E2 -22362.867} C_VEL
LIN {X 0,Y 230.121,Z 878.183,A -85,B 0,C 180,E1 -22364.624,E2 -22364.624} C_VEL
LIN {X 0,Y 229.979,Z 878.594,A -85,B 0,C 180,E1 -22365.343,E2 -22365.343} C_VEL
LIN {X 0,Y 229.425,Z 879.689,A -85,B 0,C 180,E1 -22366.576,E2 -22366.576} C_VEL
LIN {X 0,Y 227.868,Z 881.678,A -85,B 0,C 180,E1 -22367.752,E2 -22367.752} C_VEL
LIN {X 0,Y 222.472,Z 888.133,A -85,B 0,C 180,E1 -22370.816,E2 -22370.816} C_VEL
LIN {X 0,Y 217.55,Z 893.565,A -85,B 0,C 180,E1 -22373.298,E2 -22373.298} C_VEL
LIN {X 0,Y 212.025,Z 898.852,A -85,B 0,C 180,E1 -22375.702,E2 -22375.702} C_VEL
LIN {X 0,Y 204.5,Z 904.995,A -85,B 0,C 180,E1 -22378.969,E2 -22378.969} C_VEL
LIN {X 0,Y 197.561,Z 910.143,A -85,B 0,C 180,E1 -22382.795,E2 -22382.795} C_VEL
LIN {X 0,Y 192.73,Z 913.381,A -85,B 0,C 180,E1 -22386.352,E2 -22386.352} C_VEL
LIN {X 0,Y 188.635,Z 915.706,A -85,B 0,C 180,E1 -22390.408,E2 -22390.408} C_VEL
LIN {X 0,Y 185.669,Z 916.788,A -85,B 0,C 180,E1 -22394.635,E2 -22394.635} C_VEL
LIN {X 0,Y 184.131,Z 916.631,A -85,B 0,C 180,E1 -22398.998,E2 -22398.998} C_VEL
LIN {X 0,Y 183.812,Z 915.028,A -85,B 0,C 180,E1 -22403.79,E2 -22403.79} C_VEL
LIN {X 0,Y 184.252,Z 912.301,A -85,B 0,C 180,E1 -22407.814,E2 -22407.814} C_VEL
LIN {X 0,Y 184.656,Z 910.992,A -85,B 0,C 180,E1 -22409.319,E2 -22409.319} C_VEL
LIN {X 0,Y 184.34,Z 912.733,A -85,B 0,C 180,E1 -22411.042,E2 -22411.042} C_VEL
LIN {X 0,Y 183.348,Z 914.141,A -85,B 0,C 180,E1 -22412.8,E2 -22412.8} C_VEL
LIN {X 0,Y 180.213,Z 915.541,A -85,B 0,C 180,E1 -22415.732,E2 -22415.732} C_VEL
LIN {X 0,Y 177.835,Z 916.205,A -85,B 0,C 180,E1 -22418.17,E2 -22418.17} C_VEL
LIN {X 0,Y 177.004,Z 916.708,A -85,B 0,C 180,E1 -22420.07,E2 -22420.07} C_VEL
LIN {X 0,Y 177.026,Z 916.851,A -85,B 0,C 180,E1 -22420.71,E2 -22420.71} C_VEL
LIN {X 0,Y 177.802,Z 917.434,A -85,B 0,C 180,E1 -22423.719,E2 -22423.719} C_VEL
LIN {X 0,Y 180.245,Z 917.264,A -85,B 0,C 180,E1 -22428.176,E2 -22428.176} C_VEL
LIN {X 0,Y 183.941,Z 915.866,A -85,B 0,C 180,E1 -22432.463,E2 -22432.463} C_VEL
LIN {X 0,Y 188.766,Z 913.312,A -85,B 0,C 180,E1 -22436.537,E2 -22436.537} C_VEL
LIN {X 0,Y 194.908,Z 909.581,A -85,B 0,C 180,E1 -22440.319,E2 -22440.319} C_VEL
LIN {X 0,Y 200.237,Z 905.99,A -85,B 0,C 180,E1 -22442.958,E2 -22442.958} C_VEL
LIN {X 0,Y 208.359,Z 900.067,A -85,B 0,C 180,E1 -22446.177,E2 -22446.177} C_VEL
LIN {X 0,Y 212.34,Z 896.74,A -85,B 0,C 180,E1 -22447.757,E2 -22447.757} C_VEL
LIN {X 0,Y 214.103,Z 895.119,A -85,B 0,C 180,E1 -22448.586,E2 -22448.586} C_VEL
LIN {X 0,Y 217.012,Z 891.943,A -85,B 0,C 180,E1 -22450.369,E2 -22450.369} C_VEL
LIN {X 0,Y 220.21,Z 888.255,A -85,B 0,C 180,E1 -22452.771,E2 -22452.771} C_VEL
LIN {X 0,Y 221.343,Z 886.692,A -85,B 0,C 180,E1 -22454.31,E2 -22454.31} C_VEL
LIN {X 0,Y 221.931,Z 885.417,A -85,B 0,C 180,E1 -22456.749,E2 -22456.749} C_VEL
LIN {X 0,Y 222.056,Z 885.031,A -85,B 0,C 180,E1 -22459.429,E2 -22459.429} C_VEL
LIN {X 0,Y 221.943,Z 885.192,A -85,B 0,C 180,E1 -22460.703,E2 -22460.703} C_VEL
LIN {X 0,Y 221.246,Z 886.153,A -85,B 0,C 180,E1 -22462.874,E2 -22462.874} C_VEL
LIN {X 0,Y 220.461,Z 886.757,A -85,B 0,C 180,E1 -22463.24,E2 -22463.24} C_VEL
LIN {X 0,Y 210.643,Z 893.324,A -85,B 0,C 180,E1 -22466.481,E2 -22466.481} C_VEL
LIN {X 0,Y 204.44,Z 896.802,A -85,B 0,C 180,E1 -22468.957,E2 -22468.957} C_VEL
LIN {X 0,Y 197.375,Z 900.174,A -85,B 0,C 180,E1 -22472.424,E2 -22472.424} C_VEL
LIN {X 0,Y 191.171,Z 902.25,A -85,B 0,C 180,E1 -22476.145,E2 -22476.145} C_VEL
LIN {X 0,Y 186.067,Z 903.063,A -85,B 0,C 180,E1 -22480.124,E2 -22480.124} C_VEL
LIN {X 0,Y 182.102,Z 902.639,A -85,B 0,C 180,E1 -22484.324,E2 -22484.324} C_VEL
LIN {X 0,Y 179.102,Z 900.933,A -85,B 0,C 180,E1 -22488.683,E2 -22488.683} C_VEL
LIN {X 0,Y 177.403,Z 897.86,A -85,B 0,C 180,E1 -22493.172,E2 -22493.172} C_VEL
LIN {X 0,Y 176.807,Z 894.667,A -85,B 0,C 180,E1 -22496.579,E2 -22496.579} C_VEL
LIN {X 0,Y 176.508,Z 888.944,A -85,B 0,C 180,E1 -22501.138,E2 -22501.138} C_VEL
LIN {X 0,Y 176.579,Z 882.173,A -85,B 0,C 180,E1 -22505.309,E2 -22505.309} C_VEL
LIN {X 0,Y 177.197,Z 874.262,A -85,B 0,C 180,E1 -22509.126,E2 -22509.126} C_VEL
LIN {X 0,Y 178.151,Z 865.636,A -85,B 0,C 180,E1 -22512.529,E2 -22512.529} C_VEL
LIN {X 0,Y 179.544,Z 855.195,A -85,B 0,C 180,E1 -22515.9,E2 -22515.9} C_VEL
LIN {X 0,Y 181.023,Z 844.594,A -85,B 0,C 180,E1 -22518.678,E2 -22518.678} C_VEL
LIN {X 0,Y 182.308,Z 835.804,A -85,B 0,C 180,E1 -22520.593,E2 -22520.593} C_VEL
LIN {X 0,Y 183.031,Z 830.156,A -85,B 0,C 180,E1 -22521.675,E2 -22521.675} C_VEL
LIN {X 0,Y 180.907,Z 818.066,A -85,B 0,C 180,E1 -22523.755,E2 -22523.755} C_VEL
LIN {X 0,Y 178.407,Z 804.331,A -85,B 0,C 180,E1 -22525.676,E2 -22525.676} C_VEL
LIN {X 0,Y 177.471,Z 799.38,A -85,B 0,C 180,E1 -22526.295,E2 -22526.295} C_VEL
LIN {X 0,Y 177.809,Z 799.33,A -85,B 0,C 180,E1 -22530.916,E2 -22530.916} C_VEL
LIN {X 0,Y 178.142,Z 799.293,A -85,B 0,C 180,E1 -22534.056,E2 -22534.056} C_VEL
LIN {X 0,Y 178.354,Z 799.264,A -85,B 0,C 180,E1 -22539.082,E2 -22539.082} C_VEL
LIN {X 0,Y 178.388,Z 799.26,A -85,B 0,C 180,E1 -22542.044,E2 -22542.044} C_VEL
LIN {X 0,Y 178.388,Z 799.264,A -85,B 0,C 180,E1 -22545.162,E2 -22545.162} C_VEL
LIN {X 0,Y 178.397,Z 799.26,A -85,B 0,C 180,E1 -22548.457,E2 -22548.457} C_VEL
LIN {X 0,Y 178.416,Z 799.259,A -85,B 0,C 180,E1 -22553.781,E2 -22553.781} C_VEL
LIN {X 0,Y 178.477,Z 799.251,A -85,B 0,C 180,E1 -22556.545,E2 -22556.545} C_VEL
LIN {X 0,Y 178.437,Z 799.257,A -85,B 0,C 180,E1 -22561.794,E2 -22561.794} C_VEL
LIN {X 0,Y 178.508,Z 799.248,A -85,B 0,C 180,E1 -22564.888,E2 -22564.888} C_VEL
LIN {X 0,Y 178.582,Z 799.238,A -85,B 0,C 180,E1 -22570.814,E2 -22570.814} C_VEL
LIN {X 0,Y 178.638,Z 799.226,A -85,B 0,C 180,E1 -22576.346,E2 -22576.346} C_VEL
LIN {X 0,Y 178.898,Z 799.199,A -85,B 0,C 180,E1 -22580.959,E2 -22580.959} C_VEL
LIN {X 0,Y 179.114,Z 799.172,A -85,B 0,C 180,E1 -22587.751,E2 -22587.751} C_VEL
LIN {X 0,Y 179.335,Z 799.148,A -85,B 0,C 180,E1 -22590,E2 -22590} C_VEL
LIN {X 0,Y 178.818,Z 799.206,A -85,B 0,C 180,E1 -22594.508,E2 -22594.508} C_VEL
LIN {X 0,Y 178.897,Z 799.199,A -85,B 0,C 180,E1 -22599.041,E2 -22599.041} C_VEL
LIN {X 0,Y 178.635,Z 799.227,A -85,B 0,C 180,E1 -22603.654,E2 -22603.654} C_VEL
LIN {X 0,Y 178.582,Z 799.238,A -85,B 0,C 180,E1 -22609.186,E2 -22609.186} C_VEL
LIN {X 0,Y 178.508,Z 799.248,A -85,B 0,C 180,E1 -22615.112,E2 -22615.112} C_VEL
LIN {X 0,Y 178.453,Z 799.252,A -85,B 0,C 180,E1 -22620.796,E2 -22620.796} C_VEL
LIN {X 0,Y 178.477,Z 799.251,A -85,B 0,C 180,E1 -22624.22,E2 -22624.22} C_VEL
LIN {X 0,Y 178.389,Z 799.261,A -85,B 0,C 180,E1 -22629.076,E2 -22629.076} C_VEL
LIN {X 0,Y 178.392,Z 799.26,A -85,B 0,C 180,E1 -22632.047,E2 -22632.047} C_VEL
LIN {X 0,Y 178.388,Z 799.265,A -85,B 0,C 180,E1 -22635.166,E2 -22635.166} C_VEL
LIN {X 0,Y 178.395,Z 799.259,A -85,B 0,C 180,E1 -22638.463,E2 -22638.463} C_VEL
LIN {X 0,Y 178.368,Z 799.265,A -85,B 0,C 180,E1 -22642.003,E2 -22642.003} C_VEL
LIN {X 0,Y 178.167,Z 799.288,A -85,B 0,C 180,E1 -22646.482,E2 -22646.482} C_VEL
LIN {X 0,Y 177.634,Z 799.358,A -85,B 0,C 180,E1 -22651.658,E2 -22651.658} C_VEL
LIN {X 0,Y 177.49,Z 799.54,A -85,B 0,C 180,E1 -22654.142,E2 -22654.142} C_VEL
LIN {X 0,Y 180.208,Z 814.018,A -85,B 0,C 180,E1 -22656.034,E2 -22656.034} C_VEL
LIN {X 0,Y 182.57,Z 827.213,A -85,B 0,C 180,E1 -22658.184,E2 -22658.184} C_VEL
LIN {X 0,Y 182.859,Z 829.802,A -85,B 0,C 180,E1 -22658.648,E2 -22658.648} C_VEL
LIN {X 0,Y 181.233,Z 841.625,A -85,B 0,C 180,E1 -22661.051,E2 -22661.051} C_VEL
LIN {X 0,Y 179.857,Z 851.669,A -85,B 0,C 180,E1 -22663.545,E2 -22663.545} C_VEL
LIN {X 0,Y 178.378,Z 862.662,A -85,B 0,C 180,E1 -22666.909,E2 -22666.909} C_VEL
LIN {X 0,Y 177.33,Z 871.741,A -85,B 0,C 180,E1 -22670.305,E2 -22670.305} C_VEL
LIN {X 0,Y 176.694,Z 879.612,A -85,B 0,C 180,E1 -22673.921,E2 -22673.921} C_VEL
LIN {X 0,Y 176.471,Z 886.251,A -85,B 0,C 180,E1 -22677.72,E2 -22677.72} C_VEL
LIN {X 0,Y 176.556,Z 891.073,A -85,B 0,C 180,E1 -22681.143,E2 -22681.143} C_VEL
LIN {X 0,Y 176.91,Z 894.942,A -85,B 0,C 180,E1 -22684.559,E2 -22684.559} C_VEL
LIN {X 0,Y 178.004,Z 898.734,A -85,B 0,C 180,E1 -22689.089,E2 -22689.089} C_VEL
LIN {X 0,Y 180.448,Z 901.167,A -85,B 0,C 180,E1 -22693.516,E2 -22693.516} C_VEL
LIN {X 0,Y 183.741,Z 902.251,A -85,B 0,C 180,E1 -22697.82,E2 -22697.82} C_VEL
LIN {X 0,Y 188.21,Z 902.065,A -85,B 0,C 180,E1 -22701.928,E2 -22701.928} C_VEL
LIN {X 0,Y 193.921,Z 900.612,A -85,B 0,C 180,E1 -22705.781,E2 -22705.781} C_VEL
LIN {X 0,Y 200.54,Z 897.875,A -85,B 0,C 180,E1 -22709.384,E2 -22709.384} C_VEL
LIN {X 0,Y 208.142,Z 893.813,A -85,B 0,C 180,E1 -22712.702,E2 -22712.702} C_VEL
LIN {X 0,Y 216.68,Z 888.374,A -85,B 0,C 180,E1 -22715.722,E2 -22715.722} C_VEL
LIN {X 0,Y 221.144,Z 885.115,A -85,B 0,C 180,E1 -22717.146,E2 -22717.146} C_VEL
LIN {X 0,Y 222.944,Z 883.666,A -85,B 0,C 180,E1 -22717.992,E2 -22717.992} C_VEL
LIN {X 0,Y 224.11,Z 882.336,A -85,B 0,C 180,E1 -22721.192,E2 -22721.192} C_VEL
LIN {X 0,Y 224.535,Z 882.403,A -85,B 0,C 180,E1 -22723.953,E2 -22723.953} C_VEL
LIN {X 0,Y 223.506,Z 884.104,A -85,B 0,C 180,E1 -22726.323,E2 -22726.323} C_VEL
LIN {X 0,Y 218.957,Z 888.839,A -85,B 0,C 180,E1 -22728.852,E2 -22728.852} C_VEL
LIN {X 0,Y 213.956,Z 893.863,A -85,B 0,C 180,E1 -22731.383,E2 -22731.383} C_VEL
LIN {X 0,Y 208.292,Z 898.821,A -85,B 0,C 180,E1 -22733.81,E2 -22733.81} C_VEL
LIN {X 0,Y 200.387,Z 904.742,A -85,B 0,C 180,E1 -22737.07,E2 -22737.07} C_VEL
LIN {X 0,Y 193.377,Z 909.416,A -85,B 0,C 180,E1 -22740.617,E2 -22740.617} C_VEL
LIN {X 0,Y 188.828,Z 912.082,A -85,B 0,C 180,E1 -22743.472,E2 -22743.472} C_VEL
LIN {X 0,Y 183.947,Z 914.64,A -85,B 0,C 180,E1 -22747.538,E2 -22747.538} C_VEL
LIN {X 0,Y 180.26,Z 916.015,A -85,B 0,C 180,E1 -22751.826,E2 -22751.826} C_VEL
LIN {X 0,Y 177.82,Z 916.14,A -85,B 0,C 180,E1 -22756.282,E2 -22756.282} C_VEL
LIN {X 0,Y 176.83,Z 915.039,A -85,B 0,C 180,E1 -22760.852,E2 -22760.852} C_VEL
LIN {X 0,Y 176.923,Z 912.611,A -85,B 0,C 180,E1 -22765.443,E2 -22765.443} C_VEL
LIN {X 0,Y 177.734,Z 909.479,A -85,B 0,C 180,E1 -22769.363,E2 -22769.363} C_VEL
LIN {X 0,Y 177.155,Z 912.285,A -85,B 0,C 180,E1 -22772.274,E2 -22772.274} C_VEL
LIN {X 0,Y 176.697,Z 915.37,A -85,B 0,C 180,E1 -22776.853,E2 -22776.853} C_VEL
LIN {X 0,Y 177.026,Z 916.851,A -85,B 0,C 180,E1 -22780.71,E2 -22780.71} C_VEL
LIN {X 0,Y 176.82,Z 917.223,A -85,B 0,C 180,E1 -22782.616,E2 -22782.616} C_VEL
LIN {X 0,Y 175.235,Z 917.194,A -85,B 0,C 180,E1 -22785.798,E2 -22785.798} C_VEL
LIN {X 0,Y 174.309,Z 916.851,A -85,B 0,C 180,E1 -22788.378,E2 -22788.378} C_VEL
LIN {X 0,Y 174.661,Z 916.547,A -85,B 0,C 180,E1 -22790.31,E2 -22790.31} C_VEL
LIN {X 0,Y 175.086,Z 916.383,A -85,B 0,C 180,E1 -22790.938,E2 -22790.938} C_VEL
LIN {X 0,Y 179.798,Z 914.746,A -85,B 0,C 180,E1 -22795.466,E2 -22795.466} C_VEL
LIN {X 0,Y 185.541,Z 912.02,A -85,B 0,C 180,E1 -22799.5,E2 -22799.5} C_VEL
LIN {X 0,Y 192.422,Z 908.158,A -85,B 0,C 180,E1 -22803.22,E2 -22803.22} C_VEL
LIN {X 0,Y 200.608,Z 903.066,A -85,B 0,C 180,E1 -22806.553,E2 -22806.553} C_VEL
LIN {X 0,Y 206.961,Z 898.553,A -85,B 0,C 180,E1 -22808.92,E2 -22808.92} C_VEL
LIN {X 0,Y 210.336,Z 895.608,A -85,B 0,C 180,E1 -22810.659,E2 -22810.659} C_VEL
LIN {X 0,Y 213.217,Z 892.855,A -85,B 0,C 180,E1 -22812.51,E2 -22812.51} C_VEL
LIN {X 0,Y 214.481,Z 891.55,A -85,B 0,C 180,E1 -22813.482,E2 -22813.482} C_VEL
LIN {X 0,Y 215.791,Z 889.797,A -85,B 0,C 180,E1 -22815.767,E2 -22815.767} C_VEL
LIN {X 0,Y 216.154,Z 889.007,A -85,B 0,C 180,E1 -22818.402,E2 -22818.402} C_VEL
LIN {X 0,Y 216.13,Z 888.955,A -85,B 0,C 180,E1 -22819.43,E2 -22819.43} C_VEL
LIN {X 0,Y 215.552,Z 889.435,A -85,B 0,C 180,E1 -22821.719,E2 -22821.719} C_VEL
LIN {X 0,Y 213.879,Z 890.566,A -85,B 0,C 180,E1 -22822.56,E2 -22822.56} C_VEL
LIN {X 0,Y 204.808,Z 895.769,A -85,B 0,C 180,E1 -22825.514,E2 -22825.514} C_VEL
LIN {X 0,Y 198.623,Z 898.794,A -85,B 0,C 180,E1 -22827.941,E2 -22827.941} C_VEL
LIN {X 0,Y 191.256,Z 901.661,A -85,B 0,C 180,E1 -22831.462,E2 -22831.462} C_VEL
LIN {X 0,Y 184.788,Z 903.337,A -85,B 0,C 180,E1 -22835.267,E2 -22835.267} C_VEL
LIN {X 0,Y 179.459,Z 903.781,A -85,B 0,C 180,E1 -22839.36,E2 -22839.36} C_VEL
LIN {X 0,Y 175.299,Z 902.958,A -85,B 0,C 180,E1 -22843.699,E2 -22843.699} C_VEL
LIN {X 0,Y 172.157,Z 900.874,A -85,B 0,C 180,E1 -22848.22,E2 -22848.22} C_VEL
LIN {X 0,Y 170.38,Z 897.491,A -85,B 0,C 180,E1 -22852.889,E2 -22852.889} C_VEL
LIN {X 0,Y 169.758,Z 894.018,A -85,B 0,C 180,E1 -22856.437,E2 -22856.437} C_VEL
LIN {X 0,Y 169.474,Z 889.665,A -85,B 0,C 180,E1 -22859.998,E2 -22859.998} C_VEL
LIN {X 0,Y 169.464,Z 883.249,A -85,B 0,C 180,E1 -22864.159,E2 -22864.159} C_VEL
LIN {X 0,Y 170.01,Z 875.247,A -85,B 0,C 180,E1 -22868.317,E2 -22868.317} C_VEL
LIN {X 0,Y 170.898,Z 866.776,A -85,B 0,C 180,E1 -22871.863,E2 -22871.863} C_VEL
LIN {X 0,Y 172.176,Z 856.484,A -85,B 0,C 180,E1 -22875.383,E2 -22875.383} C_VEL
LIN {X 0,Y 173.823,Z 844.966,A -85,B 0,C 180,E1 -22878.564,E2 -22878.564} C_VEL
LIN {X 0,Y 175.291,Z 834.961,A -85,B 0,C 180,E1 -22880.842,E2 -22880.842} C_VEL
LIN {X 0,Y 175.896,Z 830.375,A -85,B 0,C 180,E1 -22881.755,E2 -22881.755} C_VEL
LIN {X 0,Y 173.788,Z 818.625,A -85,B 0,C 180,E1 -22883.851,E2 -22883.851} C_VEL
LIN {X 0,Y 171.2,Z 804.472,A -85,B 0,C 180,E1 -22885.902,E2 -22885.902} C_VEL
LIN {X 0,Y 170.435,Z 800.256,A -85,B 0,C 180,E1 -22886.444,E2 -22886.444} C_VEL
LIN {X 0,Y 170.721,Z 800.216,A -85,B 0,C 180,E1 -22890.174,E2 -22890.174} C_VEL
LIN {X 0,Y 171.118,Z 800.169,A -85,B 0,C 180,E1 -22895.096,E2 -22895.096} C_VEL
LIN {X 0,Y 171.303,Z 800.143,A -85,B 0,C 180,E1 -22898.784,E2 -22898.784} C_VEL
LIN {X 0,Y 171.314,Z 800.144,A -85,B 0,C 180,E1 -22904.216,E2 -22904.216} C_VEL
LIN {X 0,Y 171.329,Z 800.138,A -85,B 0,C 180,E1 -22908.979,E2 -22908.979} C_VEL
LIN {X 0,Y 171.381,Z 800.134,A -85,B 0,C 180,E1 -22912.039,E2 -22912.039} C_VEL
LIN {X 0,Y 171.392,Z 800.136,A -85,B 0,C 180,E1 -22915.091,E2 -22915.091} C_VEL
LIN {X 0,Y 171.402,Z 800.131,A -85,B 0,C 180,E1 -22920.525,E2 -22920.525} C_VEL
LIN {X 0,Y 171.433,Z 800.127,A -85,B 0,C 180,E1 -22925.798,E2 -22925.798} C_VEL
LIN {X 0,Y 171.538,Z 800.116,A -85,B 0,C 180,E1 -22930.867,E2 -22930.867} C_VEL
LIN {X 0,Y 171.552,Z 800.11,A -85,B 0,C 180,E1 -22935.771,E2 -22935.771} C_VEL
LIN {X 0,Y 171.836,Z 800.079,A -85,B 0,C 180,E1 -22940.584,E2 -22940.584} C_VEL
LIN {X 0,Y 171.773,Z 800.083,A -85,B 0,C 180,E1 -22945.306,E2 -22945.306} C_VEL
LIN {X 0,Y 172.3,Z 800.024,A -85,B 0,C 180,E1 -22950,E2 -22950} C_VEL
LIN {X 0,Y 171.849,Z 800.076,A -85,B 0,C 180,E1 -22957.047,E2 -22957.047} C_VEL
LIN {X 0,Y 171.759,Z 800.087,A -85,B 0,C 180,E1 -22960.895,E2 -22960.895} C_VEL
LIN {X 0,Y 171.514,Z 800.121,A -85,B 0,C 180,E1 -22966.669,E2 -22966.669} C_VEL
LIN {X 0,Y 171.507,Z 800.119,A -85,B 0,C 180,E1 -22969.534,E2 -22969.534} C_VEL
LIN {X 0,Y 171.437,Z 800.128,A -85,B 0,C 180,E1 -22975.6,E2 -22975.6} C_VEL
LIN {X 0,Y 171.411,Z 800.13,A -85,B 0,C 180,E1 -22980.574,E2 -22980.574} C_VEL
LIN {X 0,Y 171.386,Z 800.137,A -85,B 0,C 180,E1 -22985.036,E2 -22985.036} C_VEL
LIN {X 0,Y 171.351,Z 800.139,A -85,B 0,C 180,E1 -22988.809,E2 -22988.809} C_VEL
LIN {X 0,Y 171.315,Z 800.144,A -85,B 0,C 180,E1 -22994.219,E2 -22994.219} C_VEL
LIN {X 0,Y 171.324,Z 800.14,A -85,B 0,C 180,E1 -22998.982,E2 -22998.982} C_VEL
LIN {X 0,Y 171.317,Z 800.143,A -85,B 0,C 180,E1 -23002.026,E2 -23002.026} C_VEL
LIN {X 0,Y 171.156,Z 800.165,A -85,B 0,C 180,E1 -23005.209,E2 -23005.209} C_VEL
LIN {X 0,Y 170.737,Z 800.214,A -85,B 0,C 180,E1 -23010.402,E2 -23010.402} C_VEL
LIN {X 0,Y 170.453,Z 800.293,A -85,B 0,C 180,E1 -23013.999,E2 -23013.999} C_VEL
LIN {X 0,Y 173.124,Z 814.721,A -85,B 0,C 180,E1 -23015.959,E2 -23015.959} C_VEL
LIN {X 0,Y 175.585,Z 828.361,A -85,B 0,C 180,E1 -23018.283,E2 -23018.283} C_VEL
LIN {X 0,Y 175.777,Z 829.581,A -85,B 0,C 180,E1 -23018.509,E2 -23018.509} C_VEL
LIN {X 0,Y 174.206,Z 840.78,A -85,B 0,C 180,E1 -23020.868,E2 -23020.868} C_VEL
LIN {X 0,Y 172.646,Z 851.964,A -85,B 0,C 180,E1 -23023.75,E2 -23023.75} C_VEL
LIN {X 0,Y 171.317,Z 862.172,A -85,B 0,C 180,E1 -23026.963,E2 -23026.963} C_VEL
LIN {X 0,Y 170.234,Z 871.366,A -85,B 0,C 180,E1 -23030.497,E2 -23030.497} C_VEL
LIN {X 0,Y 169.591,Z 879.789,A -85,B 0,C 180,E1 -23034.518,E2 -23034.518} C_VEL
LIN {X 0,Y 169.427,Z 886.976,A -85,B 0,C 180,E1 -23038.814,E2 -23038.814} C_VEL
LIN {X 0,Y 169.611,Z 891.738,A -85,B 0,C 180,E1 -23042.377,E2 -23042.377} C_VEL
LIN {X 0,Y 170.266,Z 896.627,A -85,B 0,C 180,E1 -23047.116,E2 -23047.116} C_VEL
LIN {X 0,Y 172.117,Z 900.042,A -85,B 0,C 180,E1 -23051.783,E2 -23051.783} C_VEL
LIN {X 0,Y 175.155,Z 902.151,A -85,B 0,C 180,E1 -23056.314,E2 -23056.314} C_VEL
LIN {X 0,Y 179.233,Z 902.995,A -85,B 0,C 180,E1 -23060.667,E2 -23060.667} C_VEL
LIN {X 0,Y 184.556,Z 902.571,A -85,B 0,C 180,E1 -23064.767,E2 -23064.767} C_VEL
LIN {X 0,Y 191.035,Z 900.871,A -85,B 0,C 180,E1 -23068.574,E2 -23068.574} C_VEL
LIN {X 0,Y 198.373,Z 897.975,A -85,B 0,C 180,E1 -23072.104,E2 -23072.104} C_VEL
LIN {X 0,Y 206.774,Z 893.765,A -85,B 0,C 180,E1 -23075.299,E2 -23075.299} C_VEL
LIN {X 0,Y 215.917,Z 888.168,A -85,B 0,C 180,E1 -23078.204,E2 -23078.204} C_VEL
LIN {X 0,Y 217.435,Z 887.092,A -85,B 0,C 180,E1 -23079.128,E2 -23079.128} C_VEL
LIN {X 0,Y 218.501,Z 886.423,A -85,B 0,C 180,E1 -23082.492,E2 -23082.492} C_VEL
LIN {X 0,Y 218.114,Z 887.392,A -85,B 0,C 180,E1 -23085.146,E2 -23085.146} C_VEL
LIN {X 0,Y 217.516,Z 888.073,A -85,B 0,C 180,E1 -23085.853,E2 -23085.853} C_VEL
LIN {X 0,Y 212.233,Z 892.806,A -85,B 0,C 180,E1 -23088.525,E2 -23088.525} C_VEL
LIN {X 0,Y 206.753,Z 897.399,A -85,B 0,C 180,E1 -23091.034,E2 -23091.034} C_VEL
LIN {X 0,Y 200.68,Z 901.872,A -85,B 0,C 180,E1 -23093.462,E2 -23093.462} C_VEL
LIN {X 0,Y 192.609,Z 906.949,A -85,B 0,C 180,E1 -23096.816,E2 -23096.816} C_VEL
LIN {X 0,Y 185.576,Z 910.822,A -85,B 0,C 180,E1 -23100.506,E2 -23100.506} C_VEL
LIN {X 0,Y 179.813,Z 913.543,A -85,B 0,C 180,E1 -23104.536,E2 -23104.536} C_VEL
LIN {X 0,Y 175.28,Z 915.128,A -85,B 0,C 180,E1 -23108.847,E2 -23108.847} C_VEL
LIN {X 0,Y 172.011,Z 915.527,A -85,B 0,C 180,E1 -23113.381,E2 -23113.381} C_VEL
LIN {X 0,Y 170.266,Z 914.755,A -85,B 0,C 180,E1 -23118.09,E2 -23118.09} C_VEL
LIN {X 0,Y 169.874,Z 912.564,A -85,B 0,C 180,E1 -23123.196,E2 -23123.196} C_VEL
LIN {X 0,Y 170.372,Z 909.289,A -85,B 0,C 180,E1 -23127.636,E2 -23127.636} C_VEL
LIN {X 0,Y 170.836,Z 907.801,A -85,B 0,C 180,E1 -23129.411,E2 -23129.411} C_VEL
LIN {X 0,Y 170.251,Z 910.741,A -85,B 0,C 180,E1 -23132.366,E2 -23132.366} C_VEL
LIN {X 0,Y 169.785,Z 913.78,A -85,B 0,C 180,E1 -23136.546,E2 -23136.546} C_VEL
LIN {X 0,Y 170.258,Z 916.06,A -85,B 0,C 180,E1 -23141.911,E2 -23141.911} C_VEL
LIN {X 0,Y 171.989,Z 916.781,A -85,B 0,C 180,E1 -23146.621,E2 -23146.621} C_VEL
LIN {X 0,Y 175.086,Z 916.383,A -85,B 0,C 180,E1 -23150.938,E2 -23150.938} C_VEL
LIN {X 0,Y 176.115,Z 915.977,A -85,B 0,C 180,E1 -23152.832,E2 -23152.832} C_VEL
LIN {X 0,Y 176.634,Z 914.902,A -85,B 0,C 180,E1 -23156.03,E2 -23156.03} C_VEL
LIN {X 0,Y 177.835,Z 913.326,A -85,B 0,C 180,E1 -23159.156,E2 -23159.156} C_VEL
LIN {X 0,Y 179.873,Z 912.135,A -85,B 0,C 180,E1 -23160.88,E2 -23160.88} C_VEL
LIN {X 0,Y 186.561,Z 908.946,A -85,B 0,C 180,E1 -23164.407,E2 -23164.407} C_VEL
LIN {X 0,Y 195.044,Z 904.371,A -85,B 0,C 180,E1 -23167.775,E2 -23167.775} C_VEL
LIN {X 0,Y 201.634,Z 900.227,A -85,B 0,C 180,E1 -23170.153,E2 -23170.153} C_VEL
LIN {X 0,Y 205.15,Z 897.574,A -85,B 0,C 180,E1 -23171.915,E2 -23171.915} C_VEL
LIN {X 0,Y 208.122,Z 895.099,A -85,B 0,C 180,E1 -23173.809,E2 -23173.809} C_VEL
LIN {X 0,Y 209.191,Z 893.976,A -85,B 0,C 180,E1 -23175.126,E2 -23175.126} C_VEL
LIN {X 0,Y 209.999,Z 892.885,A -85,B 0,C 180,E1 -23177.415,E2 -23177.415} C_VEL
LIN {X 0,Y 209.723,Z 892.756,A -85,B 0,C 180,E1 -23180.451,E2 -23180.451} C_VEL
LIN {X 0,Y 209.506,Z 892.894,A -85,B 0,C 180,E1 -23181.096,E2 -23181.096} C_VEL
LIN {X 0,Y 201.496,Z 897.02,A -85,B 0,C 180,E1 -23183.631,E2 -23183.631} C_VEL
LIN {X 0,Y 192.838,Z 900.655,A -85,B 0,C 180,E1 -23186.858,E2 -23186.858} C_VEL
LIN {X 0,Y 185.186,Z 903.064,A -85,B 0,C 180,E1 -23190.436,E2 -23190.436} C_VEL
LIN {X 0,Y 178.445,Z 904.307,A -85,B 0,C 180,E1 -23194.325,E2 -23194.325} C_VEL
LIN {X 0,Y 172.862,Z 904.346,A -85,B 0,C 180,E1 -23198.534,E2 -23198.534} C_VEL
LIN {X 0,Y 168.496,Z 903.174,A -85,B 0,C 180,E1 -23203.022,E2 -23203.022} C_VEL
LIN {X 0,Y 165.231,Z 900.729,A -85,B 0,C 180,E1 -23207.719,E2 -23207.719} C_VEL
LIN {X 0,Y 163.361,Z 896.994,A -85,B 0,C 180,E1 -23212.582,E2 -23212.582} C_VEL
LIN {X 0,Y 162.592,Z 891.835,A -85,B 0,C 180,E1 -23217.52,E2 -23217.52} C_VEL
LIN {X 0,Y 162.417,Z 886.883,A -85,B 0,C 180,E1 -23221.237,E2 -23221.237} C_VEL
LIN {X 0,Y 162.51,Z 880.815,A -85,B 0,C 180,E1 -23224.959,E2 -23224.959} C_VEL
LIN {X 0,Y 163.116,Z 872.695,A -85,B 0,C 180,E1 -23229.026,E2 -23229.026} C_VEL
LIN {X 0,Y 163.997,Z 864.626,A -85,B 0,C 180,E1 -23232.37,E2 -23232.37} C_VEL
LIN {X 0,Y 165.428,Z 853.889,A -85,B 0,C 180,E1 -23236.027,E2 -23236.027} C_VEL
LIN {X 0,Y 166.979,Z 842.935,A -85,B 0,C 180,E1 -23239.035,E2 -23239.035} C_VEL
LIN {X 0,Y 168.508,Z 832.453,A -85,B 0,C 180,E1 -23241.401,E2 -23241.401} C_VEL
LIN {X 0,Y 168.545,Z 829.323,A -85,B 0,C 180,E1 -23242.039,E2 -23242.039} C_VEL
LIN {X 0,Y 166.114,Z 815.964,A -85,B 0,C 180,E1 -23244.428,E2 -23244.428} C_VEL
LIN {X 0,Y 163.694,Z 802.967,A -85,B 0,C 180,E1 -23246.328,E2 -23246.328} C_VEL
LIN {X 0,Y 163.419,Z 801.13,A -85,B 0,C 180,E1 -23246.563,E2 -23246.563} C_VEL
LIN {X 0,Y 163.731,Z 801.083,A -85,B 0,C 180,E1 -23251,E2 -23251} C_VEL
LIN {X 0,Y 164.073,Z 801.046,A -85,B 0,C 180,E1 -23255.525,E2 -23255.525} C_VEL
LIN {X 0,Y 164.248,Z 801.02,A -85,B 0,C 180,E1 -23259.925,E2 -23259.925} C_VEL
LIN {X 0,Y 164.275,Z 801.021,A -85,B 0,C 180,E1 -23263.34,E2 -23263.34} C_VEL
LIN {X 0,Y 164.258,Z 801.024,A -85,B 0,C 180,E1 -23266.797,E2 -23266.797} C_VEL
LIN {X 0,Y 164.289,Z 801.014,A -85,B 0,C 180,E1 -23270.35,E2 -23270.35} C_VEL
LIN {X 0,Y 164.324,Z 801.015,A -85,B 0,C 180,E1 -23274.347,E2 -23274.347} C_VEL
LIN {X 0,Y 164.36,Z 801.007,A -85,B 0,C 180,E1 -23279.128,E2 -23279.128} C_VEL
LIN {X 0,Y 164.387,Z 801.007,A -85,B 0,C 180,E1 -23284.689,E2 -23284.689} C_VEL
LIN {X 0,Y 164.431,Z 801.001,A -85,B 0,C 180,E1 -23290.095,E2 -23290.095} C_VEL
LIN {X 0,Y 164.48,Z 800.994,A -85,B 0,C 180,E1 -23295.145,E2 -23295.145} C_VEL
LIN {X 0,Y 164.757,Z 800.962,A -85,B 0,C 180,E1 -23300.176,E2 -23300.176} C_VEL
LIN {X 0,Y 164.812,Z 800.953,A -85,B 0,C 180,E1 -23302.65,E2 -23302.65} C_VEL
LIN {X 0,Y 165.264,Z 800.9,A -85,B 0,C 180,E1 -23310,E2 -23310} C_VEL
LIN {X 0,Y 164.81,Z 800.953,A -85,B 0,C 180,E1 -23317.35,E2 -23317.35} C_VEL
LIN {X 0,Y 164.694,Z 800.967,A -85,B 0,C 180,E1 -23321.059,E2 -23321.059} C_VEL
LIN {X 0,Y 164.444,Z 801,A -85,B 0,C 180,E1 -23327.408,E2 -23327.408} C_VEL
LIN {X 0,Y 164.442,Z 801,A -85,B 0,C 180,E1 -23329.993,E2 -23329.993} C_VEL
LIN {X 0,Y 164.363,Z 801.01,A -85,B 0,C 180,E1 -23336.118,E2 -23336.118} C_VEL
LIN {X 0,Y 164.346,Z 801.007,A -85,B 0,C 180,E1 -23341.216,E2 -23341.216} C_VEL
LIN {X 0,Y 164.288,Z 801.021,A -85,B 0,C 180,E1 -23346.791,E2 -23346.791} C_VEL
LIN {X 0,Y 164.285,Z 801.014,A -85,B 0,C 180,E1 -23349.918,E2 -23349.918} C_VEL
LIN {X 0,Y 164.274,Z 801.023,A -85,B 0,C 180,E1 -23353.344,E2 -23353.344} C_VEL
LIN {X 0,Y 164.257,Z 801.023,A -85,B 0,C 180,E1 -23356.801,E2 -23356.801} C_VEL
LIN {X 0,Y 164.255,Z 801.019,A -85,B 0,C 180,E1 -23360.369,E2 -23360.369} C_VEL
LIN {X 0,Y 164.136,Z 801.038,A -85,B 0,C 180,E1 -23364.444,E2 -23364.444} C_VEL
LIN {X 0,Y 163.751,Z 801.081,A -85,B 0,C 180,E1 -23369.135,E2 -23369.135} C_VEL
LIN {X 0,Y 163.433,Z 801.127,A -85,B 0,C 180,E1 -23373.872,E2 -23373.872} C_VEL
LIN {X 0,Y 166.036,Z 815.331,A -85,B 0,C 180,E1 -23375.91,E2 -23375.91} C_VEL
LIN {X 0,Y 168.423,Z 828.579,A -85,B 0,C 180,E1 -23378.266,E2 -23378.266} C_VEL
LIN {X 0,Y 168.203,Z 833.203,A -85,B 0,C 180,E1 -23379.2,E2 -23379.2} C_VEL
LIN {X 0,Y 166.564,Z 844.705,A -85,B 0,C 180,E1 -23381.872,E2 -23381.872} C_VEL
LIN {X 0,Y 164.918,Z 856.18,A -85,B 0,C 180,E1 -23385.188,E2 -23385.188} C_VEL
LIN {X 0,Y 163.838,Z 864.837,A -85,B 0,C 180,E1 -23388.246,E2 -23388.246} C_VEL
LIN {X 0,Y 162.939,Z 873.568,A -85,B 0,C 180,E1 -23391.944,E2 -23391.944} C_VEL
LIN {X 0,Y 162.405,Z 881.874,A -85,B 0,C 180,E1 -23396.281,E2 -23396.281} C_VEL
LIN {X 0,Y 162.411,Z 887.618,A -85,B 0,C 180,E1 -23400.003,E2 -23400.003} C_VEL
LIN {X 0,Y 162.664,Z 892.308,A -85,B 0,C 180,E1 -23403.718,E2 -23403.718} C_VEL
LIN {X 0,Y 163.269,Z 896.074,A -85,B 0,C 180,E1 -23407.422,E2 -23407.422} C_VEL
LIN {X 0,Y 165.186,Z 899.863,A -85,B 0,C 180,E1 -23412.285,E2 -23412.285} C_VEL
LIN {X 0,Y 168.366,Z 902.344,A -85,B 0,C 180,E1 -23416.992,E2 -23416.992} C_VEL
LIN {X 0,Y 172.641,Z 903.546,A -85,B 0,C 180,E1 -23421.495,E2 -23421.495} C_VEL
LIN {X 0,Y 178.208,Z 903.502,A -85,B 0,C 180,E1 -23425.712,E2 -23425.712} C_VEL
LIN {X 0,Y 184.955,Z 902.255,A -85,B 0,C 180,E1 -23429.605,E2 -23429.605} C_VEL
LIN {X 0,Y 192.595,Z 899.847,A -85,B 0,C 180,E1 -23433.189,E2 -23433.189} C_VEL
LIN {X 0,Y 201.272,Z 896.145,A -85,B 0,C 180,E1 -23436.415,E2 -23436.415} C_VEL
LIN {X 0,Y 210.752,Z 891.102,A -85,B 0,C 180,E1 -23439.318,E2 -23439.318} C_VEL
LIN {X 0,Y 211.783,Z 890.51,A -85,B 0,C 180,E1 -23440.248,E2 -23440.248} C_VEL
LIN {X 0,Y 212.162,Z 890.344,A -85,B 0,C 180,E1 -23441.494,E2 -23441.494} C_VEL
LIN {X 0,Y 212.376,Z 890.492,A -85,B 0,C 180,E1 -23443.278,E2 -23443.278} C_VEL
LIN {X 0,Y 212.287,Z 890.736,A -85,B 0,C 180,E1 -23444.048,E2 -23444.048} C_VEL
LIN {X 0,Y 210.82,Z 892.154,A -85,B 0,C 180,E1 -23445.567,E2 -23445.567} C_VEL
LIN {X 0,Y 203.466,Z 897.704,A -85,B 0,C 180,E1 -23448.982,E2 -23448.982} C_VEL
LIN {X 0,Y 197.268,Z 901.863,A -85,B 0,C 180,E1 -23451.43,E2 -23451.43} C_VEL
LIN {X 0,Y 186.753,Z 907.762,A -85,B 0,C 180,E1 -23455.633,E2 -23455.633} C_VEL
LIN {X 0,Y 179.461,Z 911.193,A -85,B 0,C 180,E1 -23459.396,E2 -23459.396} C_VEL
LIN {X 0,Y 173.416,Z 913.499,A -85,B 0,C 180,E1 -23463.526,E2 -23463.526} C_VEL
LIN {X 0,Y 168.666,Z 914.691,A -85,B 0,C 180,E1 -23467.975,E2 -23467.975} C_VEL
LIN {X 0,Y 165.234,Z 914.738,A -85,B 0,C 180,E1 -23472.678,E2 -23472.678} C_VEL
LIN {X 0,Y 163.371,Z 913.64,A -85,B 0,C 180,E1 -23477.579,E2 -23477.579} C_VEL
LIN {X 0,Y 162.919,Z 911.164,A -85,B 0,C 180,E1 -23482.845,E2 -23482.845} C_VEL
LIN {X 0,Y 163.474,Z 907.639,A -85,B 0,C 180,E1 -23487.536,E2 -23487.536} C_VEL
LIN {X 0,Y 163.976,Z 905.955,A -85,B 0,C 180,E1 -23489.386,E2 -23489.386} C_VEL
LIN {X 0,Y 163.369,Z 909.098,A -85,B 0,C 180,E1 -23492.466,E2 -23492.466} C_VEL
LIN {X 0,Y 162.832,Z 912.69,A -85,B 0,C 180,E1 -23497.44,E2 -23497.44} C_VEL
LIN {X 0,Y 163.363,Z 914.949,A -85,B 0,C 180,E1 -23502.422,E2 -23502.422} C_VEL
LIN {X 0,Y 165.213,Z 915.989,A -85,B 0,C 180,E1 -23507.324,E2 -23507.324} C_VEL
LIN {X 0,Y 168.654,Z 915.9,A -85,B 0,C 180,E1 -23512.027,E2 -23512.027} C_VEL
LIN {X 0,Y 173.398,Z 914.678,A -85,B 0,C 180,E1 -23516.477,E2 -23516.477} C_VEL
LIN {X 0,Y 179.42,Z 912.346,A -85,B 0,C 180,E1 -23520.612,E2 -23520.612} C_VEL
LIN {X 0,Y 179.873,Z 912.135,A -85,B 0,C 180,E1 -23520.88,E2 -23520.88} C_VEL
LIN {X 0,Y 182.154,Z 910.91,A -85,B 0,C 180,E1 -23522.559,E2 -23522.559} C_VEL
LIN {X 0,Y 187.293,Z 906.923,A -85,B 0,C 180,E1 -23527.701,E2 -23527.701} C_VEL
LIN {X 0,Y 190.023,Z 905.275,A -85,B 0,C 180,E1 -23529.196,E2 -23529.196} C_VEL
LIN {X 0,Y 191.177,Z 904.654,A -85,B 0,C 180,E1 -23529.633,E2 -23529.633} C_VEL
LIN {X 0,Y 196.403,Z 901.788,A -85,B 0,C 180,E1 -23531.453,E2 -23531.453} C_VEL
LIN {X 0,Y 200.001,Z 899.374,A -85,B 0,C 180,E1 -23533.254,E2 -23533.254} C_VEL
LIN {X 0,Y 201.586,Z 898.279,A -85,B 0,C 180,E1 -23534.209,E2 -23534.209} C_VEL
LIN {X 0,Y 203.317,Z 896.651,A -85,B 0,C 180,E1 -23536.544,E2 -23536.544} C_VEL
LIN {X 0,Y 203.521,Z 896.039,A -85,B 0,C 180,E1 -23539.439,E2 -23539.439} C_VEL
LIN {X 0,Y 203.466,Z 896.035,A -85,B 0,C 180,E1 -23540.04,E2 -23540.04} C_VEL
LIN {X 0,Y 200.903,Z 897.194,A -85,B 0,C 180,E1 -23540.971,E2 -23540.971} C_VEL
LIN {X 0,Y 191.466,Z 900.997,A -85,B 0,C 180,E1 -23544.032,E2 -23544.032} C_VEL
LIN {X 0,Y 182.998,Z 903.538,A -85,B 0,C 180,E1 -23547.473,E2 -23547.473} C_VEL
LIN {X 0,Y 175.486,Z 904.922,A -85,B 0,C 180,E1 -23551.274,E2 -23551.274} C_VEL
LIN {X 0,Y 169.075,Z 905.134,A -85,B 0,C 180,E1 -23555.436,E2 -23555.436} C_VEL
LIN {X 0,Y 163.815,Z 904.166,A -85,B 0,C 180,E1 -23559.925,E2 -23559.925} C_VEL
LIN {X 0,Y 159.963,Z 901.992,A -85,B 0,C 180,E1 -23564.713,E2 -23564.713} C_VEL
LIN {X 0,Y 157.033,Z 898.382,A -85,B 0,C 180,E1 -23569.935,E2 -23569.935} C_VEL
LIN {X 0,Y 155.876,Z 893.811,A -85,B 0,C 180,E1 -23574.824,E2 -23574.824} C_VEL
LIN {X 0,Y 155.461,Z 889.243,A -85,B 0,C 180,E1 -23578.702,E2 -23578.702} C_VEL
LIN {X 0,Y 155.407,Z 882.564,A -85,B 0,C 180,E1 -23583.238,E2 -23583.238} C_VEL
LIN {X 0,Y 155.888,Z 874.315,A -85,B 0,C 180,E1 -23587.77,E2 -23587.77} C_VEL
LIN {X 0,Y 156.785,Z 865.569,A -85,B 0,C 180,E1 -23591.634,E2 -23591.634} C_VEL
LIN {X 0,Y 158.09,Z 854.935,A -85,B 0,C 180,E1 -23595.467,E2 -23595.467} C_VEL
LIN {X 0,Y 159.634,Z 844.334,A -85,B 0,C 180,E1 -23598.611,E2 -23598.611} C_VEL
LIN {X 0,Y 161.334,Z 832.749,A -85,B 0,C 180,E1 -23601.394,E2 -23601.394} C_VEL
LIN {X 0,Y 161.404,Z 829.631,A -85,B 0,C 180,E1 -23602.056,E2 -23602.056} C_VEL
LIN {X 0,Y 158.924,Z 816.048,A -85,B 0,C 180,E1 -23604.591,E2 -23604.591} C_VEL
LIN {X 0,Y 156.819,Z 804.814,A -85,B 0,C 180,E1 -23606.321,E2 -23606.321} C_VEL
LIN {X 0,Y 156.387,Z 802.006,A -85,B 0,C 180,E1 -23606.702,E2 -23606.702} C_VEL
LIN {X 0,Y 156.76,Z 801.954,A -85,B 0,C 180,E1 -23612.544,E2 -23612.544} C_VEL
LIN {X 0,Y 157.052,Z 801.923,A -85,B 0,C 180,E1 -23616.342,E2 -23616.342} C_VEL
LIN {X 0,Y 157.164,Z 801.902,A -85,B 0,C 180,E1 -23620.518,E2 -23620.518} C_VEL
LIN {X 0,Y 157.173,Z 801.905,A -85,B 0,C 180,E1 -23625.675,E2 -23625.675} C_VEL
LIN {X 0,Y 157.221,Z 801.899,A -85,B 0,C 180,E1 -23631.257,E2 -23631.257} C_VEL
LIN {X 0,Y 157.271,Z 801.894,A -85,B 0,C 180,E1 -23634.484,E2 -23634.484} C_VEL
LIN {X 0,Y 157.273,Z 801.887,A -85,B 0,C 180,E1 -23638.102,E2 -23638.102} C_VEL
LIN {X 0,Y 157.302,Z 801.891,A -85,B 0,C 180,E1 -23643.462,E2 -23643.462} C_VEL
LIN {X 0,Y 157.37,Z 801.882,A -85,B 0,C 180,E1 -23649.683,E2 -23649.683} C_VEL
LIN {X 0,Y 157.415,Z 801.873,A -85,B 0,C 180,E1 -23654.462,E2 -23654.462} C_VEL
LIN {X 0,Y 157.68,Z 801.844,A -85,B 0,C 180,E1 -23659.73,E2 -23659.73} C_VEL
LIN {X 0,Y 157.75,Z 801.833,A -85,B 0,C 180,E1 -23662.319,E2 -23662.319} C_VEL
LIN {X 0,Y 158.226,Z 801.777,A -85,B 0,C 180,E1 -23670,E2 -23670} C_VEL
LIN {X 0,Y 157.749,Z 801.833,A -85,B 0,C 180,E1 -23677.681,E2 -23677.681} C_VEL
LIN {X 0,Y 157.624,Z 801.848,A -85,B 0,C 180,E1 -23681.228,E2 -23681.228} C_VEL
LIN {X 0,Y 157.413,Z 801.873,A -85,B 0,C 180,E1 -23685.538,E2 -23685.538} C_VEL
LIN {X 0,Y 157.349,Z 801.881,A -85,B 0,C 180,E1 -23690.936,E2 -23690.936} C_VEL
LIN {X 0,Y 157.303,Z 801.892,A -85,B 0,C 180,E1 -23696.682,E2 -23696.682} C_VEL
LIN {X 0,Y 157.258,Z 801.89,A -85,B 0,C 180,E1 -23702.432,E2 -23702.432} C_VEL
LIN {X 0,Y 157.262,Z 801.895,A -85,B 0,C 180,E1 -23706.451,E2 -23706.451} C_VEL
LIN {X 0,Y 157.187,Z 801.901,A -85,B 0,C 180,E1 -23712.119,E2 -23712.119} C_VEL
LIN {X 0,Y 157.179,Z 801.902,A -85,B 0,C 180,E1 -23717.883,E2 -23717.883} C_VEL
LIN {X 0,Y 157.13,Z 801.913,A -85,B 0,C 180,E1 -23723.619,E2 -23723.619} C_VEL
LIN {X 0,Y 156.746,Z 801.952,A -85,B 0,C 180,E1 -23728.419,E2 -23728.419} C_VEL
LIN {X 0,Y 156.404,Z 802.003,A -85,B 0,C 180,E1 -23733.761,E2 -23733.761} C_VEL
LIN {X 0,Y 159.059,Z 816.581,A -85,B 0,C 180,E1 -23735.964,E2 -23735.964} C_VEL
LIN {X 0,Y 161.271,Z 828.858,A -85,B 0,C 180,E1 -23738.261,E2 -23738.261} C_VEL
LIN {X 0,Y 161.211,Z 832.058,A -85,B 0,C 180,E1 -23738.924,E2 -23738.924} C_VEL
LIN {X 0,Y 159.405,Z 844.843,A -85,B 0,C 180,E1 -23742.027,E2 -23742.027} C_VEL
LIN {X 0,Y 157.876,Z 855.271,A -85,B 0,C 180,E1 -23745.172,E2 -23745.172} C_VEL
LIN {X 0,Y 156.583,Z 865.738,A -85,B 0,C 180,E1 -23749.006,E2 -23749.006} C_VEL
LIN {X 0,Y 155.753,Z 874.753,A -85,B 0,C 180,E1 -23753.074,E2 -23753.074} C_VEL
LIN {X 0,Y 155.388,Z 882.497,A -85,B 0,C 180,E1 -23757.41,E2 -23757.41} C_VEL
LIN {X 0,Y 155.459,Z 888.2,A -85,B 0,C 180,E1 -23761.298,E2 -23761.298} C_VEL
LIN {X 0,Y 155.819,Z 892.815,A -85,B 0,C 180,E1 -23765.178,E2 -23765.178} C_VEL
LIN {X 0,Y 157.07,Z 897.669,A -85,B 0,C 180,E1 -23770.313,E2 -23770.313} C_VEL
LIN {X 0,Y 159.832,Z 901.123,A -85,B 0,C 180,E1 -23775.3,E2 -23775.3} C_VEL
LIN {X 0,Y 163.676,Z 903.314,A -85,B 0,C 180,E1 -23780.093,E2 -23780.093} C_VEL
LIN {X 0,Y 168.766,Z 904.309,A -85,B 0,C 180,E1 -23784.612,E2 -23784.612} C_VEL
LIN {X 0,Y 175.271,Z 904.088,A -85,B 0,C 180,E1 -23788.765,E2 -23788.765} C_VEL
LIN {X 0,Y 182.769,Z 902.713,A -85,B 0,C 180,E1 -23792.573,E2 -23792.573} C_VEL
LIN {X 0,Y 191.238,Z 900.135,A -85,B 0,C 180,E1 -23796.018,E2 -23796.018} C_VEL
LIN {X 0,Y 200.642,Z 896.3,A -85,B 0,C 180,E1 -23799.089,E2 -23799.089} C_VEL
LIN {X 0,Y 205.499,Z 893.969,A -85,B 0,C 180,E1 -23800.528,E2 -23800.528} C_VEL
LIN {X 0,Y 205.877,Z 893.845,A -85,B 0,C 180,E1 -23801.322,E2 -23801.322} C_VEL
